{attribute 'Tc2GvlVarNames'}
VAR_GLOBAL
	{attribute 'OPC.UA.DA' := '1'}
	{attribute 'OPC.UA.DA.StructuredType' := '1'}
	arrScadaAlarms : ARRAY [1..222]  OF ST_AliasAlarms;	
	
	{attribute 'OPC.UA.DA' := '1'}
	{attribute 'OPC.UA.DA.StructuredType' := '1'}
	arrOPCUA_Alarms : ARRAY [1..10]  OF ST_Alarm_State_Alias;	
	
	
END_VAR
(*
VAR_GLOBAL PERSISTENT
stOperAlarmIniFileName: STRING:='Copy of Alarms_AR2000.xls 041121';
arrAlarmsOld: ARRAY [1..222] OF ST_AlarmStructure;
arrAlarmsOriginal,arrAlarms: ARRAY [1..222] OF ST_AlarmStructure :=[
( sName := 'a_bOperMaStInitSt', sClearName := '', sID := '1001', a := FALSE, b := FALSE, iGroup :=1, iSetDelay :=0, iResetDelay := 100, eResetMode := MANU, eBrakeProgram := B100, eAlarmProgram := 0, Enable := TRUE, iRepetitionNumber := 0 , iRepetitionPeriod := 10, Comment := 'Turbine Initialising', Param1 := (Set:=0, SetMin:=0, SetMax:=0,Comment:=''), Param2 := (Set:=0, SetMin:=0, SetMax:=0,Comment:='') ),
( sName := 'a_bOperMaStStopSt', sClearName := '', sID := '1002', a := FALSE, b := FALSE, iGroup :=1, iSetDelay :=0, iResetDelay := 0, eResetMode := MANU, eBrakeProgram := B100, eAlarmProgram := 0, Enable := TRUE, iRepetitionNumber := 0 , iRepetitionPeriod := 10, Comment := 'Turbine in the Stop state', Param1 := (Set:=0, SetMin:=0, SetMax:=0,Comment:=''), Param2 := (Set:=0, SetMin:=0, SetMax:=0,Comment:='') ),
( sName := 'a_bOperMaStIdleSt', sClearName := '', sID := '1003', a := FALSE, b := FALSE, iGroup :=1, iSetDelay :=0, iResetDelay := 0, eResetMode := MANU, eBrakeProgram := B100, eAlarmProgram := 0, Enable := TRUE, iRepetitionNumber := 0 , iRepetitionPeriod := 10, Comment := 'Turbine in the Idle state', Param1 := (Set:=0, SetMin:=0, SetMax:=0,Comment:=''), Param2 := (Set:=0, SetMin:=0, SetMax:=0,Comment:='') ),
( sName := 'a_bOperMaStStandbySt', sClearName := '', sID := '1004', a := FALSE, b := FALSE, iGroup :=1, iSetDelay :=0, iResetDelay := 0, eResetMode := MANU, eBrakeProgram := B100, eAlarmProgram := 0, Enable := TRUE, iRepetitionNumber := 0 , iRepetitionPeriod := 10, Comment := 'Turbine in the Ready state', Param1 := (Set:=0, SetMin:=0, SetMax:=0,Comment:=''), Param2 := (Set:=0, SetMin:=0, SetMax:=0,Comment:='') ),
( sName := 'a_bOperMaStPowerProductionSt', sClearName := '', sID := '1005', a := FALSE, b := FALSE, iGroup :=1, iSetDelay :=0, iResetDelay := 0, eResetMode := MANU, eBrakeProgram := B100, eAlarmProgram := 0, Enable := TRUE, iRepetitionNumber := 0 , iRepetitionPeriod := 10, Comment := 'Turbine in the Power Production state', Param1 := (Set:=0, SetMin:=0, SetMax:=0,Comment:=''), Param2 := (Set:=0, SetMin:=0, SetMax:=0,Comment:='') ),
( sName := 'a_bOperMaStNormalStopSt', sClearName := '', sID := '1006', a := FALSE, b := FALSE, iGroup :=1, iSetDelay :=0, iResetDelay := 0, eResetMode := MANU, eBrakeProgram := B100, eAlarmProgram := 0, Enable := TRUE, iRepetitionNumber := 0 , iRepetitionPeriod := 10, Comment := 'Turbine in the Normal Stop state', Param1 := (Set:=0, SetMin:=0, SetMax:=0,Comment:=''), Param2 := (Set:=0, SetMin:=0, SetMax:=0,Comment:='') ),
( sName := 'a_bOperMaStEmergencyStopSt', sClearName := '', sID := '1007', a := FALSE, b := FALSE, iGroup :=1, iSetDelay :=0, iResetDelay := 0, eResetMode := MANU, eBrakeProgram := B100, eAlarmProgram := 0, Enable := TRUE, iRepetitionNumber := 0 , iRepetitionPeriod := 10, Comment := 'Turbine in the Emergency Stop state', Param1 := (Set:=0, SetMin:=0, SetMax:=0,Comment:=''), Param2 := (Set:=0, SetMin:=0, SetMax:=0,Comment:='') ),
( sName := 'a_bOperAutostartCmdActive', sClearName := '', sID := '1008', a := FALSE, b := FALSE, iGroup :=1, iSetDelay :=0, iResetDelay := 0, eResetMode := MANU, eBrakeProgram := B99, eAlarmProgram := 0, Enable := TRUE, iRepetitionNumber := 0 , iRepetitionPeriod := 0, Comment := 'System generation inhibit removed by operator', Param1 := (Set:=0, SetMin:=0, SetMax:=0,Comment:=''), Param2 := (Set:=0, SetMin:=0, SetMax:=0,Comment:='') ),
( sName := 'a_bOperTestIdlingShutdown', sClearName := '', sID := '1009', a := FALSE, b := FALSE, iGroup :=1, iSetDelay :=0, iResetDelay := 0, eResetMode := MANU, eBrakeProgram := B17, eAlarmProgram := 0, Enable := TRUE, iRepetitionNumber := 0 , iRepetitionPeriod := 0, Comment := 'Test B17 go to Idle or Standby', Param1 := (Set:=0, SetMin:=0, SetMax:=0,Comment:=''), Param2 := (Set:=0, SetMin:=0, SetMax:=0,Comment:='') ),
( sName := 'a_bOperTestBrakingShutdown', sClearName := '', sID := '1010', a := FALSE, b := FALSE, iGroup :=1, iSetDelay :=0, iResetDelay := 0, eResetMode := MANU, eBrakeProgram := B14, eAlarmProgram := 0, Enable := TRUE, iRepetitionNumber := 0 , iRepetitionPeriod := 0, Comment := 'Test B14 apply parking brake', Param1 := (Set:=0, SetMin:=0, SetMax:=0,Comment:=''), Param2 := (Set:=0, SetMin:=0, SetMax:=0,Comment:='') ),
( sName := 'a_bOperTestSafetyVCTripShutdown', sClearName := '', sID := '1011', a := FALSE, b := FALSE, iGroup :=1, iSetDelay :=0, iResetDelay := 0, eResetMode := MANU, eBrakeProgram := B100, eAlarmProgram := 0, Enable := TRUE, iRepetitionNumber := 0 , iRepetitionPeriod := 0, Comment := 'Test B9 trip vacuum contactor', Param1 := (Set:=0, SetMin:=0, SetMax:=0,Comment:=''), Param2 := (Set:=0, SetMin:=0, SetMax:=0,Comment:='') ),
( sName := 'a_bOperTestSafetyBrakeShutdown', sClearName := '', sID := '1012', a := FALSE, b := FALSE, iGroup :=1, iSetDelay :=0, iResetDelay := 0, eResetMode := MANU, eBrakeProgram := B100, eAlarmProgram := 0, Enable := TRUE, iRepetitionNumber := 0 , iRepetitionPeriod := 0, Comment := 'Test B5 apply safety brake', Param1 := (Set:=0, SetMin:=0, SetMax:=0,Comment:=''), Param2 := (Set:=0, SetMin:=0, SetMax:=0,Comment:='') ),
( sName := 'a_bOperCmdNormalShutdownToStop', sClearName := 'Turbine manual stop using main gui button', sID := '1013', a := FALSE, b := FALSE, iGroup :=1, iSetDelay :=0, iResetDelay := 0, eResetMode := MANU, eBrakeProgram := B100, eAlarmProgram := 0, Enable := TRUE, iRepetitionNumber := 0 , iRepetitionPeriod := 0, Comment := 'Manual stop command', Param1 := (Set:=0, SetMin:=0, SetMax:=0,Comment:=''), Param2 := (Set:=0, SetMin:=0, SetMax:=0,Comment:='') ),
( sName := 'a_bOperCmdNormalShutdownToStandby', sClearName := '', sID := '1014', a := FALSE, b := FALSE, iGroup :=1, iSetDelay :=0, iResetDelay := 0, eResetMode := MANU, eBrakeProgram := B100, eAlarmProgram := 0, Enable := TRUE, iRepetitionNumber := 0 , iRepetitionPeriod := 0, Comment := '', Param1 := (Set:=0, SetMin:=0, SetMax:=0,Comment:=''), Param2 := (Set:=0, SetMin:=0, SetMax:=0,Comment:='') ),
( sName := 'a_bOperRepeatingAlarm', sClearName := '', sID := '1015', a := FALSE, b := FALSE, iGroup :=1, iSetDelay :=10, iResetDelay := 0, eResetMode := MANU, eBrakeProgram := B100, eAlarmProgram := 0, Enable := TRUE, iRepetitionNumber := 0 , iRepetitionPeriod := 10, Comment := 'Alarm which occur with this one has occured too many times', Param1 := (Set:=0, SetMin:=0, SetMax:=0,Comment:=''), Param2 := (Set:=0, SetMin:=0, SetMax:=0,Comment:='') ),
( sName := 'a_bOperResetTooLongPushed', sClearName := 'Reset Button ', sID := '1016', a := FALSE, b := FALSE, iGroup :=1, iSetDelay :=10, iResetDelay := 0, eResetMode := MANU, eBrakeProgram := B99, eAlarmProgram := 0, Enable := TRUE, iRepetitionNumber := 0 , iRepetitionPeriod := 10, Comment := 'Reset button pressed too long', Param1 := (Set:=0, SetMin:=0, SetMax:=0,Comment:=''), Param2 := (Set:=0, SetMin:=0, SetMax:=0,Comment:='') ),
( sName := 'a_bOperAlarmParameterChanged', sClearName := 'Alarm Parameter ', sID := '1017', a := FALSE, b := FALSE, iGroup :=1, iSetDelay :=0, iResetDelay := 5, eResetMode := MANU, eBrakeProgram := B99, eAlarmProgram := 0, Enable := TRUE, iRepetitionNumber := 0 , iRepetitionPeriod := 10, Comment := 'Alarm parameter has been changed', Param1 := (Set:=0, SetMin:=0, SetMax:=0,Comment:=''), Param2 := (Set:=0, SetMin:=0, SetMax:=0,Comment:='') ),
( sName := 'a_bOperIniParameterChanged', sClearName := 'Ini Parameter ', sID := '1018', a := FALSE, b := FALSE, iGroup :=1, iSetDelay :=0, iResetDelay := 5, eResetMode := MANU, eBrakeProgram := B99, eAlarmProgram := 0, Enable := TRUE, iRepetitionNumber := 0 , iRepetitionPeriod := 10, Comment := 'Ini parameter has been changed', Param1 := (Set:=0, SetMin:=0, SetMax:=0,Comment:=''), Param2 := (Set:=0, SetMin:=0, SetMax:=0,Comment:='') ),
( sName := 'a_bOperSystemReboot', sClearName := 'System ', sID := '1019', a := FALSE, b := FALSE, iGroup :=1, iSetDelay :=10, iResetDelay := 150, eResetMode := MANU, eBrakeProgram := B100, eAlarmProgram := 0, Enable := TRUE, iRepetitionNumber := 0 , iRepetitionPeriod := 10, Comment := 'System is rebooted', Param1 := (Set:=0, SetMin:=0, SetMax:=0,Comment:=''), Param2 := (Set:=0, SetMin:=0, SetMax:=0,Comment:='') ),
( sName := 'a_bOperSystemRestart ', sClearName := 'System ', sID := '1020', a := FALSE, b := FALSE, iGroup :=1, iSetDelay :=10, iResetDelay := 150, eResetMode := MANU, eBrakeProgram := B100, eAlarmProgram := 0, Enable := TRUE, iRepetitionNumber := 0 , iRepetitionPeriod := 10, Comment := 'System is restarted', Param1 := (Set:=0, SetMin:=0, SetMax:=0,Comment:=''), Param2 := (Set:=0, SetMin:=0, SetMax:=0,Comment:='') ),
( sName := 'a_bOperScopeViewNotActive', sClearName := 'ScopeView running', sID := '1021', a := FALSE, b := FALSE, iGroup :=1, iSetDelay :=100, iResetDelay := 0, eResetMode := MANU, eBrakeProgram := B17, eAlarmProgram := 0, Enable := TRUE, iRepetitionNumber := 0 , iRepetitionPeriod := 10, Comment := 'Fastlog system not active', Param1 := (Set:=0, SetMin:=0, SetMax:=0,Comment:=''), Param2 := (Set:=0, SetMin:=0, SetMax:=0,Comment:='') ),
( sName := 'a_bOperXMLDataUncertainty', sClearName := 'Turbine data XML file Ok', sID := '1022', a := FALSE, b := FALSE, iGroup :=1, iSetDelay :=0, iResetDelay := 0, eResetMode := MANU, eBrakeProgram := B17, eAlarmProgram := 0, Enable := TRUE, iRepetitionNumber := 0 , iRepetitionPeriod := 10, Comment := 'Turbine data XML file uncertainty', Param1 := (Set:=0, SetMin:=0, SetMax:=0,Comment:=''), Param2 := (Set:=0, SetMin:=0, SetMax:=0,Comment:='') ),
( sName := 'a_bOperSoftwareUpdate', sClearName := 'System software ', sID := '1023', a := FALSE, b := FALSE, iGroup :=1, iSetDelay :=0, iResetDelay := 0, eResetMode := MANU, eBrakeProgram := B17, eAlarmProgram := 0, Enable := FALSE, iRepetitionNumber := 0 , iRepetitionPeriod := 10, Comment := 'System software is updated', Param1 := (Set:=0, SetMin:=0, SetMax:=0,Comment:=''), Param2 := (Set:=0, SetMin:=0, SetMax:=0,Comment:='') ),
( sName := 'a_bOperFastlogComsErr', sClearName := 'a_bOperLossOfCommsToArrayController', sID := '1024', a := FALSE, b := FALSE, iGroup :=1, iSetDelay :=0, iResetDelay := 0, eResetMode := MANU, eBrakeProgram := B99, eAlarmProgram := 0, Enable := TRUE, iRepetitionNumber := 0 , iRepetitionPeriod := 10, Comment := 'Loss of Comms with ARL Array PLC', Param1 := (Set:=0, SetMin:=0, SetMax:=0,Comment:=''), Param2 := (Set:=0, SetMin:=0, SetMax:=0,Comment:='') ),
( sName := 'a_bOperInOffMode', sClearName := 'Turbine in OFF Mode', sID := '1025', a := FALSE, b := FALSE, iGroup :=1, iSetDelay :=0, iResetDelay := 0, eResetMode := MANU, eBrakeProgram := B100, eAlarmProgram := 0, Enable := TRUE, iRepetitionNumber := 0 , iRepetitionPeriod := 10, Comment := 'Turbine entering OFF Mode', Param1 := (Set:=0, SetMin:=0, SetMax:=0,Comment:=''), Param2 := (Set:=0, SetMin:=0, SetMax:=0,Comment:='') ),
( sName := 'a_bOperInServiceMode', sClearName := 'Turbine in Service Mode', sID := '1026', a := FALSE, b := FALSE, iGroup :=1, iSetDelay :=0, iResetDelay := 0, eResetMode := MANU, eBrakeProgram := B100, eAlarmProgram := 0, Enable := TRUE, iRepetitionNumber := 0 , iRepetitionPeriod := 10, Comment := 'Turbine entering Service Mode', Param1 := (Set:=0, SetMin:=0, SetMax:=0,Comment:=''), Param2 := (Set:=0, SetMin:=0, SetMax:=0,Comment:='') ),
( sName := 'a_bOperInAutomaticMode', sClearName := 'Turbine in Automatic Mode', sID := '1027', a := FALSE, b := FALSE, iGroup :=1, iSetDelay :=0, iResetDelay := 0, eResetMode := MANU, eBrakeProgram := B100, eAlarmProgram := 0, Enable := TRUE, iRepetitionNumber := 0 , iRepetitionPeriod := 10, Comment := 'Turbine entering Automatic Mode', Param1 := (Set:=0, SetMin:=0, SetMax:=0,Comment:=''), Param2 := (Set:=0, SetMin:=0, SetMax:=0,Comment:='') ),
( sName := 'a_bOperInManualMode', sClearName := 'Turbine in Manual Mode', sID := '1028', a := FALSE, b := FALSE, iGroup :=1, iSetDelay :=0, iResetDelay := 0, eResetMode := MANU, eBrakeProgram := B100, eAlarmProgram := 0, Enable := TRUE, iRepetitionNumber := 0 , iRepetitionPeriod := 10, Comment := 'Turbine entering Manual Mode', Param1 := (Set:=0, SetMin:=0, SetMax:=0,Comment:=''), Param2 := (Set:=0, SetMin:=0, SetMax:=0,Comment:='') ),
( sName := 'a_bOperInFATMode', sClearName := 'Turbine in Factory Acceptance Test Nautilus Mode', sID := '1029', a := FALSE, b := FALSE, iGroup :=1, iSetDelay :=0, iResetDelay := 0, eResetMode := MANU, eBrakeProgram := B100, eAlarmProgram := 0, Enable := TRUE, iRepetitionNumber := 0 , iRepetitionPeriod := 10, Comment := 'Turbine entering Factory Acceptance Test Nautilus Mode', Param1 := (Set:=0, SetMin:=0, SetMax:=0,Comment:=''), Param2 := (Set:=0, SetMin:=0, SetMax:=0,Comment:='') ),
( sName := 'a_bHydairFaultActive', sClearName := 'Cleared', sID := '1030', a := FALSE, b := FALSE, iGroup :=1, iSetDelay :=0, iResetDelay := 0, eResetMode := MANU, eBrakeProgram := B99, eAlarmProgram := 0, Enable := TRUE, iRepetitionNumber := 0 , iRepetitionPeriod := 0, Comment := '', Param1 := (Set:=0, SetMin:=0, SetMax:=0,Comment:=''), Param2 := (Set:=0, SetMin:=0, SetMax:=0,Comment:='') ),
( sName := 'a_bHydairOfflineFilterClogged', sClearName := 'Cleared', sID := '1031', a := FALSE, b := FALSE, iGroup :=1, iSetDelay :=0, iResetDelay := 0, eResetMode := MANU, eBrakeProgram := B99, eAlarmProgram := 0, Enable := TRUE, iRepetitionNumber := 0 , iRepetitionPeriod := 0, Comment := '', Param1 := (Set:=0, SetMin:=0, SetMax:=0,Comment:=''), Param2 := (Set:=0, SetMin:=0, SetMax:=0,Comment:='') ),
( sName := 'a_bMainReturnPressureFilterClogged', sClearName := 'Cleared', sID := '1032', a := FALSE, b := FALSE, iGroup :=1, iSetDelay :=0, iResetDelay := 0, eResetMode := MANU, eBrakeProgram := B99, eAlarmProgram := 0, Enable := TRUE, iRepetitionNumber := 0 , iRepetitionPeriod := 0, Comment := '', Param1 := (Set:=0, SetMin:=0, SetMax:=0,Comment:=''), Param2 := (Set:=0, SetMin:=0, SetMax:=0,Comment:='') ),
( sName := 'a_bMainSupplyPressureFilterClogged', sClearName := 'Cleared', sID := '1033', a := FALSE, b := FALSE, iGroup :=1, iSetDelay :=0, iResetDelay := 0, eResetMode := MANU, eBrakeProgram := B99, eAlarmProgram := 0, Enable := TRUE, iRepetitionNumber := 0 , iRepetitionPeriod := 0, Comment := '', Param1 := (Set:=0, SetMin:=0, SetMax:=0,Comment:=''), Param2 := (Set:=0, SetMin:=0, SetMax:=0,Comment:='') ),
( sName := 'a_bHydairPassiveCtrlState', sClearName := 'Cleared', sID := '1034', a := FALSE, b := FALSE, iGroup :=1, iSetDelay :=0, iResetDelay := 0, eResetMode := MANU, eBrakeProgram := B99, eAlarmProgram := 0, Enable := TRUE, iRepetitionNumber := 0 , iRepetitionPeriod := 0, Comment := '', Param1 := (Set:=0, SetMin:=0, SetMax:=0,Comment:=''), Param2 := (Set:=0, SetMin:=0, SetMax:=0,Comment:='') ),
( sName := 'a_bHydairStartUp', sClearName := 'Cleared', sID := '1035', a := FALSE, b := FALSE, iGroup :=1, iSetDelay :=0, iResetDelay := 0, eResetMode := MANU, eBrakeProgram := B99, eAlarmProgram := 0, Enable := TRUE, iRepetitionNumber := 0 , iRepetitionPeriod := 0, Comment := '', Param1 := (Set:=0, SetMin:=0, SetMax:=0,Comment:=''), Param2 := (Set:=0, SetMin:=0, SetMax:=0,Comment:='') ),
( sName := 'a_bHydairReadyToOperate', sClearName := 'Cleared', sID := '1036', a := FALSE, b := FALSE, iGroup :=1, iSetDelay :=0, iResetDelay := 0, eResetMode := MANU, eBrakeProgram := B99, eAlarmProgram := 0, Enable := TRUE, iRepetitionNumber := 0 , iRepetitionPeriod := 0, Comment := '', Param1 := (Set:=0, SetMin:=0, SetMax:=0,Comment:=''), Param2 := (Set:=0, SetMin:=0, SetMax:=0,Comment:='') ),
( sName := 'a_bHydairActiveCtrlState', sClearName := 'Cleared', sID := '1037', a := FALSE, b := FALSE, iGroup :=1, iSetDelay :=0, iResetDelay := 0, eResetMode := MANU, eBrakeProgram := B99, eAlarmProgram := 0, Enable := TRUE, iRepetitionNumber := 0 , iRepetitionPeriod := 0, Comment := '', Param1 := (Set:=0, SetMin:=0, SetMax:=0,Comment:=''), Param2 := (Set:=0, SetMin:=0, SetMax:=0,Comment:='') ),
( sName := 'a_bHydairStopped', sClearName := 'Cleared', sID := '1038', a := FALSE, b := FALSE, iGroup :=1, iSetDelay :=0, iResetDelay := 0, eResetMode := MANU, eBrakeProgram := B99, eAlarmProgram := 0, Enable := TRUE, iRepetitionNumber := 0 , iRepetitionPeriod := 0, Comment := '', Param1 := (Set:=0, SetMin:=0, SetMax:=0,Comment:=''), Param2 := (Set:=0, SetMin:=0, SetMax:=0,Comment:='') ),
( sName := 'a_bHydairEstopActive', sClearName := 'Cleared', sID := '1039', a := FALSE, b := FALSE, iGroup :=1, iSetDelay :=0, iResetDelay := 0, eResetMode := MANU, eBrakeProgram := B99, eAlarmProgram := 0, Enable := TRUE, iRepetitionNumber := 0 , iRepetitionPeriod := 0, Comment := '', Param1 := (Set:=0, SetMin:=0, SetMax:=0,Comment:=''), Param2 := (Set:=0, SetMin:=0, SetMax:=0,Comment:='') ),
( sName := 'a_bHydairOilTempTooHigh', sClearName := 'Cleared', sID := '1040', a := FALSE, b := FALSE, iGroup :=1, iSetDelay :=0, iResetDelay := 0, eResetMode := MANU, eBrakeProgram := B99, eAlarmProgram := 0, Enable := TRUE, iRepetitionNumber := 0 , iRepetitionPeriod := 0, Comment := '', Param1 := (Set:=0, SetMin:=0, SetMax:=0,Comment:=''), Param2 := (Set:=0, SetMin:=0, SetMax:=0,Comment:='') ),
( sName := 'a_bHydairReadyToStartup', sClearName := 'Cleared', sID := '1041', a := FALSE, b := FALSE, iGroup :=1, iSetDelay :=0, iResetDelay := 0, eResetMode := MANU, eBrakeProgram := B99, eAlarmProgram := 0, Enable := TRUE, iRepetitionNumber := 0 , iRepetitionPeriod := 0, Comment := '', Param1 := (Set:=0, SetMin:=0, SetMax:=0,Comment:=''), Param2 := (Set:=0, SetMin:=0, SetMax:=0,Comment:='') ),
( sName := 'a_bOperRequestStopLATSystem', sClearName := 'Cleared', sID := '1042', a := FALSE, b := FALSE, iGroup :=1, iSetDelay :=0, iResetDelay := 0, eResetMode := MANU, eBrakeProgram := B99, eAlarmProgram := 0, Enable := TRUE, iRepetitionNumber := 0 , iRepetitionPeriod := 0, Comment := '', Param1 := (Set:=0, SetMin:=0, SetMax:=0,Comment:=''), Param2 := (Set:=0, SetMin:=0, SetMax:=0,Comment:='') ),
( sName := 'a_bOperRequestStartupHydair', sClearName := 'Cleared', sID := '1043', a := FALSE, b := FALSE, iGroup :=1, iSetDelay :=0, iResetDelay := 0, eResetMode := MANU, eBrakeProgram := B99, eAlarmProgram := 0, Enable := TRUE, iRepetitionNumber := 0 , iRepetitionPeriod := 0, Comment := '', Param1 := (Set:=0, SetMin:=0, SetMax:=0,Comment:=''), Param2 := (Set:=0, SetMin:=0, SetMax:=0,Comment:='') ),
( sName := 'a_bOperRequestPassivePitchCtrl', sClearName := 'Cleared', sID := '1044', a := FALSE, b := FALSE, iGroup :=1, iSetDelay :=0, iResetDelay := 0, eResetMode := MANU, eBrakeProgram := B99, eAlarmProgram := 0, Enable := TRUE, iRepetitionNumber := 0 , iRepetitionPeriod := 0, Comment := '', Param1 := (Set:=0, SetMin:=0, SetMax:=0,Comment:=''), Param2 := (Set:=0, SetMin:=0, SetMax:=0,Comment:='') ),
( sName := 'a_bOperRequestActiveLoadCtrlMode', sClearName := 'Cleared', sID := '1045', a := FALSE, b := FALSE, iGroup :=1, iSetDelay :=0, iResetDelay := 0, eResetMode := MANU, eBrakeProgram := B99, eAlarmProgram := 0, Enable := TRUE, iRepetitionNumber := 0 , iRepetitionPeriod := 0, Comment := '', Param1 := (Set:=0, SetMin:=0, SetMax:=0,Comment:=''), Param2 := (Set:=0, SetMin:=0, SetMax:=0,Comment:='') ),
( sName := 'a_bOperRequestLoadProfileStream', sClearName := 'Cleared', sID := '1046', a := FALSE, b := FALSE, iGroup :=1, iSetDelay :=0, iResetDelay := 0, eResetMode := MANU, eBrakeProgram := B99, eAlarmProgram := 0, Enable := TRUE, iRepetitionNumber := 0 , iRepetitionPeriod := 0, Comment := '', Param1 := (Set:=0, SetMin:=0, SetMax:=0,Comment:=''), Param2 := (Set:=0, SetMin:=0, SetMax:=0,Comment:='') ),
( sName := 'a_bOperLoadProfileStreamingStarted', sClearName := 'Cleared', sID := '1047', a := FALSE, b := FALSE, iGroup :=1, iSetDelay :=0, iResetDelay := 0, eResetMode := MANU, eBrakeProgram := B99, eAlarmProgram := 0, Enable := TRUE, iRepetitionNumber := 0 , iRepetitionPeriod := 0, Comment := '', Param1 := (Set:=0, SetMin:=0, SetMax:=0,Comment:=''), Param2 := (Set:=0, SetMin:=0, SetMax:=0,Comment:='') ),
( sName := 'a_bOperLoadProfilePaused', sClearName := 'Cleared', sID := '1048', a := FALSE, b := FALSE, iGroup :=1, iSetDelay :=0, iResetDelay := 0, eResetMode := MANU, eBrakeProgram := B99, eAlarmProgram := 0, Enable := TRUE, iRepetitionNumber := 0 , iRepetitionPeriod := 0, Comment := '', Param1 := (Set:=0, SetMin:=0, SetMax:=0,Comment:=''), Param2 := (Set:=0, SetMin:=0, SetMax:=0,Comment:='') ),
( sName := 'a_bOperLoadProfileFrequencyError', sClearName := 'Cleared', sID := '1049', a := FALSE, b := FALSE, iGroup :=1, iSetDelay :=0, iResetDelay := 0, eResetMode := MANU, eBrakeProgram := B99, eAlarmProgram := 0, Enable := TRUE, iRepetitionNumber := 0 , iRepetitionPeriod := 0, Comment := '', Param1 := (Set:=0, SetMin:=0, SetMax:=0,Comment:=''), Param2 := (Set:=0, SetMin:=0, SetMax:=0,Comment:='') ),
( sName := 'a_bOperPitch100HrRuntime', sClearName := 'Cleared', sID := '1050', a := FALSE, b := FALSE, iGroup :=1, iSetDelay :=0, iResetDelay := 0, eResetMode := MANU, eBrakeProgram := B99, eAlarmProgram := 0, Enable := TRUE, iRepetitionNumber := 0 , iRepetitionPeriod := 0, Comment := '', Param1 := (Set:=0, SetMin:=0, SetMax:=0,Comment:=''), Param2 := (Set:=0, SetMin:=0, SetMax:=0,Comment:='') ),
( sName := 'a_bOperB20PitchNormalShutdownCmd', sClearName := 'Cleared', sID := '1051', a := FALSE, b := FALSE, iGroup :=1, iSetDelay :=0, iResetDelay := 0, eResetMode := MANU, eBrakeProgram := B20, eAlarmProgram := 0, Enable := TRUE, iRepetitionNumber := 0 , iRepetitionPeriod := 0, Comment := '', Param1 := (Set:=0, SetMin:=0, SetMax:=0,Comment:=''), Param2 := (Set:=0, SetMin:=0, SetMax:=0,Comment:='') ),
( sName := 'a_bHydraulicsLoadMzRam1HiWarning', sClearName := 'Hydraulic Load Hi Warning', sID := '1045', a := FALSE, b := FALSE, iGroup :=1, iSetDelay :=0, iResetDelay := 0, eResetMode := MANU, eBrakeProgram := B20, eAlarmProgram := 0, Enable := TRUE, iRepetitionNumber := 0 , iRepetitionPeriod := 0, Comment := 'Hydraulic Load Hi Warning', Param1 := (Set:=450000, SetMin:=1, SetMax:=600000,Comment:='Nm'), Param2 := (Set:=1000, SetMin:=1, SetMax:=600000,Comment:='Nm') ),
( sName := 'a_bHydraulicsLoadMzRam1HiHiAlarm', sClearName := 'Hydraulic Load Hi Alarm', sID := '1046', a := FALSE, b := FALSE, iGroup :=1, iSetDelay :=0, iResetDelay := 0, eResetMode := MANU, eBrakeProgram := B1, eAlarmProgram := 0, Enable := TRUE, iRepetitionNumber := 0 , iRepetitionPeriod := 0, Comment := 'Hydraulic Load Hi Alarm', Param1 := (Set:=500000, SetMin:=1, SetMax:=600000,Comment:='Nm'), Param2 := (Set:=1000, SetMin:=1, SetMax:=600000,Comment:='Nm') ),
( sName := 'a_bHydraulicsLoadMyRam2HiWarning', sClearName := 'Hydraulic Load Hi Warning', sID := '1047', a := FALSE, b := FALSE, iGroup :=1, iSetDelay :=0, iResetDelay := 0, eResetMode := MANU, eBrakeProgram := B20, eAlarmProgram := 0, Enable := TRUE, iRepetitionNumber := 0 , iRepetitionPeriod := 0, Comment := 'Hydraulic Load Hi Warning', Param1 := (Set:=450000, SetMin:=1, SetMax:=600000,Comment:='Nm'), Param2 := (Set:=1000, SetMin:=1, SetMax:=600000,Comment:='Nm') ),
( sName := 'a_bHydraulicsLoadMyRam2HiHiAlarm', sClearName := 'Hydraulic Load Hi Alarm', sID := '1048', a := FALSE, b := FALSE, iGroup :=1, iSetDelay :=0, iResetDelay := 0, eResetMode := MANU, eBrakeProgram := B1, eAlarmProgram := 0, Enable := TRUE, iRepetitionNumber := 0 , iRepetitionPeriod := 0, Comment := 'Hydraulic Load Hi Alarm', Param1 := (Set:=500000, SetMin:=1, SetMax:=600000,Comment:='Nm'), Param2 := (Set:=1000, SetMin:=1, SetMax:=600000,Comment:='Nm') ),
( sName := 'a_bHydraulicsLoadTrackingMzRAM1Warning', sClearName := 'Hydraulic Load Control Tracking Warning', sID := '1049', a := FALSE, b := FALSE, iGroup :=1, iSetDelay :=10, iResetDelay := 10, eResetMode := MANU, eBrakeProgram := B99, eAlarmProgram := 0, Enable := TRUE, iRepetitionNumber := 0 , iRepetitionPeriod := 0, Comment := 'Hydraulic Load Control Tracking Warning', Param1 := (Set:=5, SetMin:=0, SetMax:=100,Comment:=''), Param2 := (Set:=2, SetMin:=0, SetMax:=100,Comment:='') ),
( sName := 'a_bHydraulicsLoadTrackingMzRAM1Alarm', sClearName := 'Hydraulic Load Control Tracking Alarm', sID := '1050', a := FALSE, b := FALSE, iGroup :=1, iSetDelay :=10, iResetDelay := 10, eResetMode := MANU, eBrakeProgram := B20, eAlarmProgram := 0, Enable := TRUE, iRepetitionNumber := 0 , iRepetitionPeriod := 0, Comment := 'Hydraulic Load Control Tracking Alarm', Param1 := (Set:=10, SetMin:=0, SetMax:=100,Comment:=''), Param2 := (Set:=5, SetMin:=0, SetMax:=100,Comment:='') ),
( sName := 'a_bHydraulicsLoadTrackingMyRAM2Warning', sClearName := 'Hydraulic Load Control Tracking Warning', sID := '1051', a := FALSE, b := FALSE, iGroup :=1, iSetDelay :=10, iResetDelay := 10, eResetMode := MANU, eBrakeProgram := B99, eAlarmProgram := 0, Enable := TRUE, iRepetitionNumber := 0 , iRepetitionPeriod := 0, Comment := 'Hydraulic Load Control Tracking Warning', Param1 := (Set:=5, SetMin:=0, SetMax:=100,Comment:=''), Param2 := (Set:=2, SetMin:=0, SetMax:=100,Comment:='') ),
( sName := 'a_bHydraulicsLoadTrackingMyRAM2Alarm', sClearName := 'Hydraulic Load Control Tracking Alarm', sID := '1052', a := FALSE, b := FALSE, iGroup :=1, iSetDelay :=10, iResetDelay := 10, eResetMode := MANU, eBrakeProgram := B20, eAlarmProgram := 0, Enable := TRUE, iRepetitionNumber := 0 , iRepetitionPeriod := 0, Comment := 'Hydraulic Load Control Tracking Alarm', Param1 := (Set:=10, SetMin:=0, SetMax:=100,Comment:=''), Param2 := (Set:=5, SetMin:=0, SetMax:=100,Comment:='') ),
( sName := 'a_bHydraulicsLVDTSensor1Failure', sClearName := 'Hydraulics LVDT Sensor1 Failure', sID := '1053', a := FALSE, b := FALSE, iGroup :=1, iSetDelay :=0, iResetDelay := 10, eResetMode := MANU, eBrakeProgram := B99, eAlarmProgram := 0, Enable := TRUE, iRepetitionNumber := 0 , iRepetitionPeriod := , Comment := 'Hydraulics LVDT Sensor1 Failure', Param1 := (Set:=0, SetMin:=0, SetMax:=0,Comment:=''), Param2 := (Set:=0, SetMin:=0, SetMax:=0,Comment:='') ),
( sName := 'a_bHydraulicsLVDTSensor2Failure', sClearName := 'Hydraulics LVDT Sensor2 Failure', sID := '1054', a := FALSE, b := FALSE, iGroup :=1, iSetDelay :=0, iResetDelay := 10, eResetMode := MANU, eBrakeProgram := B99, eAlarmProgram := 0, Enable := TRUE, iRepetitionNumber := 0 , iRepetitionPeriod := , Comment := 'Hydraulics LVDT Sensor2 Failure', Param1 := (Set:=0, SetMin:=0, SetMax:=0,Comment:=''), Param2 := (Set:=0, SetMin:=0, SetMax:=0,Comment:='') ),
( sName := 'a_bHydraulicsLVDTSensor3Failure', sClearName := 'Hydraulics LVDT Sensor3 Failure', sID := '1055', a := FALSE, b := FALSE, iGroup :=1, iSetDelay :=0, iResetDelay := 10, eResetMode := MANU, eBrakeProgram := B99, eAlarmProgram := 0, Enable := TRUE, iRepetitionNumber := 0 , iRepetitionPeriod := , Comment := 'Hydraulics LVDT Sensor3 Failure', Param1 := (Set:=0, SetMin:=0, SetMax:=0,Comment:=''), Param2 := (Set:=0, SetMin:=0, SetMax:=0,Comment:='') ),
( sName := 'a_bHydraulicsLVDTSensor4Failure', sClearName := 'Hydraulics LVDT Sensor4 Failure', sID := '1056', a := FALSE, b := FALSE, iGroup :=1, iSetDelay :=0, iResetDelay := 10, eResetMode := MANU, eBrakeProgram := B99, eAlarmProgram := 0, Enable := TRUE, iRepetitionNumber := 0 , iRepetitionPeriod := , Comment := 'Hydraulics LVDT Sensor4 Failure', Param1 := (Set:=0, SetMin:=0, SetMax:=0,Comment:=''), Param2 := (Set:=0, SetMin:=0, SetMax:=0,Comment:='') ),
( sName := 'a_bHydraulicsLVDTSensor5Failure', sClearName := 'Hydraulics LVDT Sensor5 Failure', sID := '1057', a := FALSE, b := FALSE, iGroup :=1, iSetDelay :=0, iResetDelay := 10, eResetMode := MANU, eBrakeProgram := B99, eAlarmProgram := 0, Enable := TRUE, iRepetitionNumber := 0 , iRepetitionPeriod := , Comment := 'Hydraulics LVDT Sensor5 Failure', Param1 := (Set:=0, SetMin:=0, SetMax:=0,Comment:=''), Param2 := (Set:=0, SetMin:=0, SetMax:=0,Comment:='') ),
( sName := 'a_bHydraulicsLVDTSensor6Failure', sClearName := 'Hydraulics LVDT Sensor6 Failure', sID := '1058', a := FALSE, b := FALSE, iGroup :=1, iSetDelay :=0, iResetDelay := 10, eResetMode := MANU, eBrakeProgram := B99, eAlarmProgram := 0, Enable := TRUE, iRepetitionNumber := 0 , iRepetitionPeriod := , Comment := 'Hydraulics LVDT Sensor6 Failure', Param1 := (Set:=0, SetMin:=0, SetMax:=0,Comment:=''), Param2 := (Set:=0, SetMin:=0, SetMax:=0,Comment:='') ),
( sName := 'a_bHydraulicsLVDTSensor7Failure', sClearName := 'Hydraulics LVDT Sensor7 Failure', sID := '1059', a := FALSE, b := FALSE, iGroup :=1, iSetDelay :=0, iResetDelay := 10, eResetMode := MANU, eBrakeProgram := B99, eAlarmProgram := 0, Enable := TRUE, iRepetitionNumber := 0 , iRepetitionPeriod := , Comment := 'Hydraulics LVDT Sensor7 Failure', Param1 := (Set:=0, SetMin:=0, SetMax:=0,Comment:=''), Param2 := (Set:=0, SetMin:=0, SetMax:=0,Comment:='') ),
( sName := 'a_bHydraulicsLVDTSensor8Failure', sClearName := 'Hydraulics LVDT Sensor8 Failure', sID := '1060', a := FALSE, b := FALSE, iGroup :=1, iSetDelay :=0, iResetDelay := 10, eResetMode := MANU, eBrakeProgram := B99, eAlarmProgram := 0, Enable := TRUE, iRepetitionNumber := 0 , iRepetitionPeriod := , Comment := 'Hydraulics LVDT Sensor8 Failure', Param1 := (Set:=0, SetMin:=0, SetMax:=0,Comment:=''), Param2 := (Set:=0, SetMin:=0, SetMax:=0,Comment:='') ),
( sName := 'a_bHydraulicsMzStrainGaugeFailure', sClearName := 'Hydraulics Mz Strain Gauge Failure', sID := '1061', a := FALSE, b := FALSE, iGroup :=1, iSetDelay :=0, iResetDelay := 10, eResetMode := MANU, eBrakeProgram := B20, eAlarmProgram := 0, Enable := TRUE, iRepetitionNumber := 0 , iRepetitionPeriod := , Comment := 'a_bHydraulicsMzStrainGaugeFailure', Param1 := (Set:=0, SetMin:=0, SetMax:=0,Comment:=''), Param2 := (Set:=0, SetMin:=0, SetMax:=0,Comment:='') ),
( sName := 'a_bHydraulicsMzStrainGaugeFailure', sClearName := 'Hydraulics Mz Strain Gauge Failure', sID := '1062', a := FALSE, b := FALSE, iGroup :=1, iSetDelay :=0, iResetDelay := 10, eResetMode := MANU, eBrakeProgram := B20, eAlarmProgram := 0, Enable := TRUE, iRepetitionNumber := 0 , iRepetitionPeriod := , Comment := 'a_bHydraulicsMzStrainGaugeFailure', Param1 := (Set:=0, SetMin:=0, SetMax:=0,Comment:=''), Param2 := (Set:=0, SetMin:=0, SetMax:=0,Comment:='') ),
( sName := 'a_bSafetyCommsLossToSSB', sClearName := '', sID := '2001', a := FALSE, b := FALSE, iGroup :=2, iSetDelay :=0, iResetDelay := 0, eResetMode := MANU, eBrakeProgram := B4, eAlarmProgram := 0, Enable := TRUE, iRepetitionNumber := 0 , iRepetitionPeriod := 0, Comment := '', Param1 := (Set:=0, SetMin:=0, SetMax:=0,Comment:=''), Param2 := (Set:=0, SetMin:=0, SetMax:=0,Comment:='') ),
( sName := 'a_bSafetyEPO_Main_Panel', sClearName := '', sID := '2002', a := FALSE, b := FALSE, iGroup :=2, iSetDelay :=0, iResetDelay := 0, eResetMode := MANU, eBrakeProgram := B1, eAlarmProgram := 0, Enable := TRUE, iRepetitionNumber := 0 , iRepetitionPeriod := 0, Comment := '', Param1 := (Set:=0, SetMin:=0, SetMax:=0,Comment:=''), Param2 := (Set:=0, SetMin:=0, SetMax:=0,Comment:='') ),
( sName := 'a_bSafetyEPO_REMOTE', sClearName := '', sID := '2003', a := FALSE, b := FALSE, iGroup :=2, iSetDelay :=0, iResetDelay := 0, eResetMode := MANU, eBrakeProgram := B1, eAlarmProgram := 0, Enable := TRUE, iRepetitionNumber := 0 , iRepetitionPeriod := 0, Comment := '', Param1 := (Set:=0, SetMin:=0, SetMax:=0,Comment:=''), Param2 := (Set:=0, SetMin:=0, SetMax:=0,Comment:='') ),
( sName := 'a_bSafetyEPO_SCADA', sClearName := '', sID := '2004', a := FALSE, b := FALSE, iGroup :=2, iSetDelay :=0, iResetDelay := 0, eResetMode := MANU, eBrakeProgram := B1, eAlarmProgram := 0, Enable := TRUE, iRepetitionNumber := 0 , iRepetitionPeriod := 0, Comment := '', Param1 := (Set:=0, SetMin:=0, SetMax:=0,Comment:=''), Param2 := (Set:=0, SetMin:=0, SetMax:=0,Comment:='') ),
( sName := 'a_bSafetyEPO_TCP', sClearName := '', sID := '2005', a := FALSE, b := FALSE, iGroup :=2, iSetDelay :=0, iResetDelay := 0, eResetMode := MANU, eBrakeProgram := B1, eAlarmProgram := 0, Enable := TRUE, iRepetitionNumber := 0 , iRepetitionPeriod := 0, Comment := '', Param1 := (Set:=0, SetMin:=0, SetMax:=0,Comment:=''), Param2 := (Set:=0, SetMin:=0, SetMax:=0,Comment:='') ),
( sName := 'a_bSafetyOperatorRequestB1', sClearName := '', sID := '2006', a := FALSE, b := FALSE, iGroup :=2, iSetDelay :=0, iResetDelay := 0, eResetMode := MANU, eBrakeProgram := B1, eAlarmProgram := 0, Enable := TRUE, iRepetitionNumber := 0 , iRepetitionPeriod := 0, Comment := '', Param1 := (Set:=0, SetMin:=0, SetMax:=0,Comment:=''), Param2 := (Set:=0, SetMin:=0, SetMax:=0,Comment:='') ),
( sName := 'a_bSafetyOperatorRequestB4', sClearName := '', sID := '2007', a := FALSE, b := FALSE, iGroup :=2, iSetDelay :=0, iResetDelay := 0, eResetMode := MANU, eBrakeProgram := B4, eAlarmProgram := 0, Enable := TRUE, iRepetitionNumber := 0 , iRepetitionPeriod := 0, Comment := '', Param1 := (Set:=0, SetMin:=0, SetMax:=0,Comment:=''), Param2 := (Set:=0, SetMin:=0, SetMax:=0,Comment:='') ),
( sName := 'a_bSafetyOperatorRequestB9', sClearName := '', sID := '2008', a := FALSE, b := FALSE, iGroup :=2, iSetDelay :=0, iResetDelay := 0, eResetMode := MANU, eBrakeProgram := B9, eAlarmProgram := 0, Enable := TRUE, iRepetitionNumber := 0 , iRepetitionPeriod := 0, Comment := '', Param1 := (Set:=0, SetMin:=0, SetMax:=0,Comment:=''), Param2 := (Set:=0, SetMin:=0, SetMax:=0,Comment:='') ),
( sName := 'a_bSafetyEncoderPositionNOTValid', sClearName := '', sID := '2009', a := FALSE, b := FALSE, iGroup :=2, iSetDelay :=0, iResetDelay := 0, eResetMode := MANU, eBrakeProgram := B1, eAlarmProgram := 0, Enable := TRUE, iRepetitionNumber := 0 , iRepetitionPeriod := 0, Comment := '', Param1 := (Set:=0, SetMin:=0, SetMax:=0,Comment:=''), Param2 := (Set:=0, SetMin:=0, SetMax:=0,Comment:='') ),
( sName := 'a_bSafetyEncoderGroupError', sClearName := '', sID := '2010', a := FALSE, b := FALSE, iGroup :=2, iSetDelay :=0, iResetDelay := 0, eResetMode := MANU, eBrakeProgram := B1, eAlarmProgram := 0, Enable := TRUE, iRepetitionNumber := 0 , iRepetitionPeriod := 0, Comment := '', Param1 := (Set:=0, SetMin:=0, SetMax:=0,Comment:=''), Param2 := (Set:=0, SetMin:=0, SetMax:=0,Comment:='') ),
( sName := 'a_bSafetyIOGroupError', sClearName := '', sID := '2011', a := FALSE, b := FALSE, iGroup :=2, iSetDelay :=0, iResetDelay := 0, eResetMode := MANU, eBrakeProgram := B1, eAlarmProgram := 0, Enable := TRUE, iRepetitionNumber := 0 , iRepetitionPeriod := 0, Comment := '', Param1 := (Set:=0, SetMin:=0, SetMax:=0,Comment:=''), Param2 := (Set:=0, SetMin:=0, SetMax:=0,Comment:='') ),
( sName := 'a_bSafetyAngInGroupError', sClearName := '', sID := '2012', a := FALSE, b := FALSE, iGroup :=2, iSetDelay :=0, iResetDelay := 0, eResetMode := MANU, eBrakeProgram := B1, eAlarmProgram := 0, Enable := TRUE, iRepetitionNumber := 0 , iRepetitionPeriod := 0, Comment := '', Param1 := (Set:=0, SetMin:=0, SetMax:=0,Comment:=''), Param2 := (Set:=0, SetMin:=0, SetMax:=0,Comment:='') ),
( sName := 'a_bSafetyPresetGroupError', sClearName := '', sID := '2013', a := FALSE, b := FALSE, iGroup :=2, iSetDelay :=0, iResetDelay := 0, eResetMode := MANU, eBrakeProgram := B1, eAlarmProgram := 0, Enable := TRUE, iRepetitionNumber := 0 , iRepetitionPeriod := 0, Comment := '', Param1 := (Set:=0, SetMin:=0, SetMax:=0,Comment:=''), Param2 := (Set:=0, SetMin:=0, SetMax:=0,Comment:='') ),
( sName := 'a_bSafetySLS_GroupError', sClearName := '', sID := '2014', a := FALSE, b := FALSE, iGroup :=2, iSetDelay :=0, iResetDelay := 0, eResetMode := MANU, eBrakeProgram := B1, eAlarmProgram := 0, Enable := TRUE, iRepetitionNumber := 0 , iRepetitionPeriod := 0, Comment := '', Param1 := (Set:=0, SetMin:=0, SetMax:=0,Comment:=''), Param2 := (Set:=0, SetMin:=0, SetMax:=0,Comment:='') ),
( sName := 'a_bSafetyX10_PNOZ_GroupError', sClearName := '', sID := '2015', a := FALSE, b := FALSE, iGroup :=2, iSetDelay :=0, iResetDelay := 0, eResetMode := MANU, eBrakeProgram := B1, eAlarmProgram := 0, Enable := TRUE, iRepetitionNumber := 0 , iRepetitionPeriod := 0, Comment := '', Param1 := (Set:=0, SetMin:=0, SetMax:=0,Comment:=''), Param2 := (Set:=0, SetMin:=0, SetMax:=0,Comment:='') ),
( sName := 'a_bSafetyX6_ExtremFine_GroupError', sClearName := '', sID := '2016', a := FALSE, b := FALSE, iGroup :=2, iSetDelay :=0, iResetDelay := 0, eResetMode := MANU, eBrakeProgram := B1, eAlarmProgram := 0, Enable := TRUE, iRepetitionNumber := 0 , iRepetitionPeriod := 0, Comment := '', Param1 := (Set:=0, SetMin:=0, SetMax:=0,Comment:=''), Param2 := (Set:=0, SetMin:=0, SetMax:=0,Comment:='') ),
( sName := 'a_bSafetyX5_EFC_GroupError', sClearName := '', sID := '2017', a := FALSE, b := FALSE, iGroup :=2, iSetDelay :=0, iResetDelay := 0, eResetMode := MANU, eBrakeProgram := B4, eAlarmProgram := 0, Enable := TRUE, iRepetitionNumber := 0 , iRepetitionPeriod := 0, Comment := '', Param1 := (Set:=0, SetMin:=0, SetMax:=0,Comment:=''), Param2 := (Set:=0, SetMin:=0, SetMax:=0,Comment:='') ),
( sName := 'a_bSafetyFBError', sClearName := '', sID := '2018', a := FALSE, b := FALSE, iGroup :=2, iSetDelay :=0, iResetDelay := 0, eResetMode := MANU, eBrakeProgram := B1, eAlarmProgram := 0, Enable := TRUE, iRepetitionNumber := 0 , iRepetitionPeriod := 0, Comment := '', Param1 := (Set:=0, SetMin:=0, SetMax:=0,Comment:=''), Param2 := (Set:=0, SetMin:=0, SetMax:=0,Comment:='') ),
( sName := 'a_bSafetyCommError', sClearName := '', sID := '2019', a := FALSE, b := FALSE, iGroup :=2, iSetDelay :=0, iResetDelay := 0, eResetMode := MANU, eBrakeProgram := B1, eAlarmProgram := 0, Enable := TRUE, iRepetitionNumber := 0 , iRepetitionPeriod := 0, Comment := '', Param1 := (Set:=0, SetMin:=0, SetMax:=0,Comment:=''), Param2 := (Set:=0, SetMin:=0, SetMax:=0,Comment:='') ),
( sName := 'a_bSafetyOutError', sClearName := '', sID := '2020', a := FALSE, b := FALSE, iGroup :=2, iSetDelay :=0, iResetDelay := 0, eResetMode := MANU, eBrakeProgram := B1, eAlarmProgram := 0, Enable := TRUE, iRepetitionNumber := 0 , iRepetitionPeriod := 0, Comment := '', Param1 := (Set:=0, SetMin:=0, SetMax:=0,Comment:=''), Param2 := (Set:=0, SetMin:=0, SetMax:=0,Comment:='') ),
( sName := 'a_bSafetyOperatorPushButtonEstopTrip', sClearName := '', sID := '2021', a := FALSE, b := FALSE, iGroup :=2, iSetDelay :=0, iResetDelay := 0, eResetMode := MANU, eBrakeProgram := B1, eAlarmProgram := 0, Enable := TRUE, iRepetitionNumber := 0 , iRepetitionPeriod := 0, Comment := '', Param1 := (Set:=0, SetMin:=0, SetMax:=0,Comment:=''), Param2 := (Set:=0, SetMin:=0, SetMax:=0,Comment:='') ),
( sName := 'a_bSafetyHydairSystemEstopTrip', sClearName := '', sID := '2022', a := FALSE, b := FALSE, iGroup :=2, iSetDelay :=0, iResetDelay := 0, eResetMode := MANU, eBrakeProgram := B1, eAlarmProgram := 0, Enable := TRUE, iRepetitionNumber := 0 , iRepetitionPeriod := 0, Comment := '', Param1 := (Set:=0, SetMin:=0, SetMax:=0,Comment:=''), Param2 := (Set:=0, SetMin:=0, SetMax:=0,Comment:='') ),
( sName := 'a_bSafetyPTCSActivatedEstopTrip_ComssLossHydair', sClearName := '', sID := '2023', a := FALSE, b := FALSE, iGroup :=2, iSetDelay :=0, iResetDelay := 0, eResetMode := MANU, eBrakeProgram := B1, eAlarmProgram := 0, Enable := TRUE, iRepetitionNumber := 0 , iRepetitionPeriod := 0, Comment := '', Param1 := (Set:=0, SetMin:=0, SetMax:=0,Comment:=''), Param2 := (Set:=0, SetMin:=0, SetMax:=0,Comment:='') ),
( sName := 'a_bSafetyPTCSActivatedEstopTrip_ExcessiveLoadTestRig', sClearName := '', sID := '2024', a := FALSE, b := FALSE, iGroup :=2, iSetDelay :=0, iResetDelay := 0, eResetMode := MANU, eBrakeProgram := B1, eAlarmProgram := 0, Enable := TRUE, iRepetitionNumber := 0 , iRepetitionPeriod := 0, Comment := '', Param1 := (Set:=0, SetMin:=0, SetMax:=0,Comment:=''), Param2 := (Set:=0, SetMin:=0, SetMax:=0,Comment:='') ),
( sName := 'a_bSafetyPitchSystemEFCActivated', sClearName := '', sID := '2025', a := FALSE, b := FALSE, iGroup :=2, iSetDelay :=0, iResetDelay := 0, eResetMode := MANU, eBrakeProgram := B4, eAlarmProgram := 0, Enable := TRUE, iRepetitionNumber := 0 , iRepetitionPeriod := 0, Comment := '', Param1 := (Set:=0, SetMin:=0, SetMax:=0,Comment:=''), Param2 := (Set:=0, SetMin:=0, SetMax:=0,Comment:='') ),
( sName := 'a_bSafetyEstopResetReq', sClearName := '', sID := '2026', a := FALSE, b := FALSE, iGroup :=2, iSetDelay :=0, iResetDelay := 0, eResetMode := MANU, eBrakeProgram := B99, eAlarmProgram := 0, Enable := TRUE, iRepetitionNumber := 0 , iRepetitionPeriod := 0, Comment := '', Param1 := (Set:=0, SetMin:=0, SetMax:=0,Comment:=''), Param2 := (Set:=0, SetMin:=0, SetMax:=0,Comment:='') ),
( sName := 'a_bSafetyEFCResetReq', sClearName := '', sID := '2027', a := FALSE, b := FALSE, iGroup :=2, iSetDelay :=0, iResetDelay := 0, eResetMode := MANU, eBrakeProgram := B99, eAlarmProgram := 0, Enable := TRUE, iRepetitionNumber := 0 , iRepetitionPeriod := 0, Comment := '', Param1 := (Set:=0, SetMin:=0, SetMax:=0,Comment:=''), Param2 := (Set:=0, SetMin:=0, SetMax:=0,Comment:='') ),
( sName := 'a_bSafetyEstopChainClosed', sClearName := '', sID := '2028', a := FALSE, b := FALSE, iGroup :=2, iSetDelay :=0, iResetDelay := 0, eResetMode := MANU, eBrakeProgram := B99, eAlarmProgram := 0, Enable := TRUE, iRepetitionNumber := 0 , iRepetitionPeriod := 0, Comment := '', Param1 := (Set:=0, SetMin:=0, SetMax:=0,Comment:=''), Param2 := (Set:=0, SetMin:=0, SetMax:=0,Comment:='') ),
( sName := 'a_bSafetyPitchEFCChainClosed', sClearName := '', sID := '2029', a := FALSE, b := FALSE, iGroup :=2, iSetDelay :=0, iResetDelay := 0, eResetMode := MANU, eBrakeProgram := B99, eAlarmProgram := 0, Enable := TRUE, iRepetitionNumber := 0 , iRepetitionPeriod := 0, Comment := '', Param1 := (Set:=0, SetMin:=0, SetMax:=0,Comment:=''), Param2 := (Set:=0, SetMin:=0, SetMax:=0,Comment:='') ),
( sName := 'a_bConverterHeartbeatFailure', sClearName := 'Heartbeat profibus', sID := '3901', a := FALSE, b := FALSE, iGroup :=3, iSetDelay :=10, iResetDelay := 0, eResetMode := MANU, eBrakeProgram := B9, eAlarmProgram := EMAIL, Enable := FALSE, iRepetitionNumber := 0 , iRepetitionPeriod := 10, Comment := 'Heartbeat failed', Param1 := (Set:=0, SetMin:=0, SetMax:=0,Comment:=''), Param2 := (Set:=0, SetMin:=0, SetMax:=0,Comment:='') ),
( sName := 'a_bSSB_NoEFCFromTC', sClearName := 'Water level below slip ring tripped low sensor', sID := '4001', a := FALSE, b := FALSE, iGroup :=4, iSetDelay :=0, iResetDelay := 0, eResetMode := MANU, eBrakeProgram := B4, eAlarmProgram := 0, Enable := TRUE, iRepetitionNumber := 0 , iRepetitionPeriod := 0, Comment := '', Param1 := (Set:=2, SetMin:=1, SetMax:=2,Comment:=''), Param2 := (Set:=0, SetMin:=0, SetMax:=0,Comment:='') ),
( sName := 'a_bSSB_bWatchDogFromPLC', sClearName := 'bWatchDogFromPLC', sID := '4002', a := FALSE, b := FALSE, iGroup :=4, iSetDelay :=0, iResetDelay := 0, eResetMode := MANU, eBrakeProgram := B4, eAlarmProgram := 0, Enable := TRUE, iRepetitionNumber := 0 , iRepetitionPeriod := 0, Comment := '', Param1 := (Set:=0, SetMin:=0, SetMax:=0,Comment:=''), Param2 := (Set:=0, SetMin:=0, SetMax:=0,Comment:='') ),
( sName := 'a_bSSB_bAllBladesAtLimit', sClearName := 'bAllBladesAtLimit', sID := '4003', a := FALSE, b := FALSE, iGroup :=4, iSetDelay :=0, iResetDelay := 0, eResetMode := MANU, eBrakeProgram := B99, eAlarmProgram := 0, Enable := TRUE, iRepetitionNumber := 0 , iRepetitionPeriod := 0, Comment := '', Param1 := (Set:=0, SetMin:=0, SetMax:=0,Comment:=''), Param2 := (Set:=0, SetMin:=0, SetMax:=0,Comment:='') ),
( sName := 'a_bSSB_bAllBladesAtFeather', sClearName := 'bAllBladesAtFeather', sID := '4004', a := FALSE, b := FALSE, iGroup :=4, iSetDelay :=0, iResetDelay := 0, eResetMode := MANU, eBrakeProgram := B99, eAlarmProgram := 0, Enable := TRUE, iRepetitionNumber := 0 , iRepetitionPeriod := 0, Comment := '', Param1 := (Set:=0, SetMin:=0, SetMax:=0,Comment:=''), Param2 := (Set:=0, SetMin:=0, SetMax:=0,Comment:='') ),
( sName := 'a_bSSB_BusOK', sClearName := 'a_bSSB_BusOK', sID := '4005', a := FALSE, b := FALSE, iGroup :=4, iSetDelay :=0, iResetDelay := 0, eResetMode := MANU, eBrakeProgram := B99, eAlarmProgram := 0, Enable := TRUE, iRepetitionNumber := 0 , iRepetitionPeriod := 0, Comment := '', Param1 := (Set:=0, SetMin:=0, SetMax:=0,Comment:=''), Param2 := (Set:=0, SetMin:=0, SetMax:=0,Comment:='') ),
( sName := 'a_bSSB_bCriticalError', sClearName := 'a_bCriticalError', sID := '4006', a := FALSE, b := FALSE, iGroup :=4, iSetDelay :=0, iResetDelay := 0, eResetMode := MANU, eBrakeProgram := B4, eAlarmProgram := 0, Enable := TRUE, iRepetitionNumber := 0 , iRepetitionPeriod := 0, Comment := '', Param1 := (Set:=0, SetMin:=0, SetMax:=0,Comment:=''), Param2 := (Set:=0, SetMin:=0, SetMax:=0,Comment:='') ),
( sName := 'a_bSSB_bFatalError', sClearName := 'a_bFatalError', sID := '4007', a := FALSE, b := FALSE, iGroup :=4, iSetDelay :=0, iResetDelay := 0, eResetMode := MANU, eBrakeProgram := B4, eAlarmProgram := 0, Enable := TRUE, iRepetitionNumber := 0 , iRepetitionPeriod := 0, Comment := '', Param1 := (Set:=0, SetMin:=0, SetMax:=0,Comment:=''), Param2 := (Set:=0, SetMin:=0, SetMax:=0,Comment:='') ),
( sName := 'a_bSSB_bReferencingFailed', sClearName := 'bReferencingFailed', sID := '4008', a := FALSE, b := FALSE, iGroup :=4, iSetDelay :=0, iResetDelay := 0, eResetMode := MANU, eBrakeProgram := B99, eAlarmProgram := 0, Enable := TRUE, iRepetitionNumber := 0 , iRepetitionPeriod := 0, Comment := '', Param1 := (Set:=0, SetMin:=0, SetMax:=0,Comment:=''), Param2 := (Set:=0, SetMin:=0, SetMax:=0,Comment:='') ),
( sName := 'a_bSSB_ExtDI1_Lube1Flt', sClearName := 'a_ExtDI1_Lube1Flt', sID := '4009', a := FALSE, b := FALSE, iGroup :=4, iSetDelay :=0, iResetDelay := 0, eResetMode := MANU, eBrakeProgram := B99, eAlarmProgram := 0, Enable := TRUE, iRepetitionNumber := 0 , iRepetitionPeriod := 0, Comment := '', Param1 := (Set:=0, SetMin:=0, SetMax:=0,Comment:=''), Param2 := (Set:=0, SetMin:=0, SetMax:=0,Comment:='') ),
( sName := 'a_bSSB_PPA_EFC1_by_Error', sClearName := 'a_PPA_EFC1_by_Error', sID := '4010', a := FALSE, b := FALSE, iGroup :=4, iSetDelay :=0, iResetDelay := 0, eResetMode := MANU, eBrakeProgram := B4, eAlarmProgram := 0, Enable := TRUE, iRepetitionNumber := 0 , iRepetitionPeriod := 0, Comment := '', Param1 := (Set:=0, SetMin:=0, SetMax:=0,Comment:=''), Param2 := (Set:=0, SetMin:=0, SetMax:=0,Comment:='') ),
( sName := 'a_bSSB_PPA_EFC1_by_bus', sClearName := 'a_PPA_EFC1_by_bus', sID := '4011', a := FALSE, b := FALSE, iGroup :=4, iSetDelay :=0, iResetDelay := 0, eResetMode := MANU, eBrakeProgram := B4, eAlarmProgram := 0, Enable := TRUE, iRepetitionNumber := 0 , iRepetitionPeriod := 0, Comment := '', Param1 := (Set:=0, SetMin:=0, SetMax:=0,Comment:=''), Param2 := (Set:=0, SetMin:=0, SetMax:=0,Comment:='') ),
( sName := 'a_bSSB_LS_active ', sClearName := 'a_PPA_EFC1_active', sID := '4012', a := FALSE, b := FALSE, iGroup :=4, iSetDelay :=0, iResetDelay := 0, eResetMode := MANU, eBrakeProgram := B99, eAlarmProgram := 0, Enable := TRUE, iRepetitionNumber := 0 , iRepetitionPeriod := 0, Comment := '', Param1 := (Set:=0, SetMin:=0, SetMax:=0,Comment:=''), Param2 := (Set:=0, SetMin:=0, SetMax:=0,Comment:='') ),
( sName := 'a_bSSB_SWLS', sClearName := 'a_bSSB_SWLS', sID := '4013', a := FALSE, b := FALSE, iGroup :=4, iSetDelay :=0, iResetDelay := 0, eResetMode := MANU, eBrakeProgram := B99, eAlarmProgram := 0, Enable := TRUE, iRepetitionNumber := 0 , iRepetitionPeriod := 0, Comment := '', Param1 := (Set:=0, SetMin:=0, SetMax:=0,Comment:=''), Param2 := (Set:=0, SetMin:=0, SetMax:=0,Comment:='') ),
( sName := 'a_bSSB_Bypass1stlimitactive', sClearName := 'a_bSSB_Bypass1stlimitactive', sID := '4014', a := FALSE, b := FALSE, iGroup :=4, iSetDelay :=0, iResetDelay := 0, eResetMode := MANU, eBrakeProgram := B99, eAlarmProgram := 0, Enable := TRUE, iRepetitionNumber := 0 , iRepetitionPeriod := 0, Comment := '', Param1 := (Set:=0, SetMin:=0, SetMax:=0,Comment:=''), Param2 := (Set:=0, SetMin:=0, SetMax:=0,Comment:='') ),
( sName := 'a_bSSB_MainsWarning', sClearName := 'Mains ok (1 = ok, 0 = general warning)', sID := '4015', a := FALSE, b := FALSE, iGroup :=4, iSetDelay :=0, iResetDelay := 0, eResetMode := MANU, eBrakeProgram := B99, eAlarmProgram := 0, Enable := TRUE, iRepetitionNumber := 0 , iRepetitionPeriod := 0, Comment := '', Param1 := (Set:=0, SetMin:=0, SetMax:=0,Comment:=''), Param2 := (Set:=0, SetMin:=0, SetMax:=0,Comment:='') ),
( sName := 'a_bSSB_CurrentBackup_heaterLow', sClearName := 'a_bSSB_CurrentBackup_heaterLow', sID := '4016', a := FALSE, b := FALSE, iGroup :=4, iSetDelay :=0, iResetDelay := 0, eResetMode := MANU, eBrakeProgram := B99, eAlarmProgram := 0, Enable := TRUE, iRepetitionNumber := 0 , iRepetitionPeriod := 0, Comment := '', Param1 := (Set:=0, SetMin:=0, SetMax:=0,Comment:=''), Param2 := (Set:=0, SetMin:=0, SetMax:=0,Comment:='') ),
( sName := 'a_bSSB_Crit_InternEncoderDeviation', sClearName := '; (motor encoder - blade encoder) > uMAX_DEVIATION', sID := '4017', a := FALSE, b := FALSE, iGroup :=4, iSetDelay :=0, iResetDelay := 0, eResetMode := MANU, eBrakeProgram := B4, eAlarmProgram := 0, Enable := TRUE, iRepetitionNumber := 0 , iRepetitionPeriod := 0, Comment := '', Param1 := (Set:=0, SetMin:=0, SetMax:=0,Comment:=''), Param2 := (Set:=0, SetMin:=0, SetMax:=0,Comment:='') ),
( sName := 'a_bSSB_Crit_ExternEncoderDeviation', sClearName := 'a_bSSB_ExternEncoderDeviation', sID := '4018', a := FALSE, b := FALSE, iGroup :=4, iSetDelay :=0, iResetDelay := 0, eResetMode := MANU, eBrakeProgram := B4, eAlarmProgram := 0, Enable := TRUE, iRepetitionNumber := 0 , iRepetitionPeriod := 0, Comment := '', Param1 := (Set:=0, SetMin:=0, SetMax:=0,Comment:=''), Param2 := (Set:=0, SetMin:=0, SetMax:=0,Comment:='') ),
( sName := 'a_bSSB_Backup_Charger_Not_Working', sClearName := '', sID := '4019', a := FALSE, b := FALSE, iGroup :=4, iSetDelay :=0, iResetDelay := 0, eResetMode := MANU, eBrakeProgram := B4, eAlarmProgram := 0, Enable := TRUE, iRepetitionNumber := 0 , iRepetitionPeriod := 0, Comment := '', Param1 := (Set:=0, SetMin:=0, SetMax:=0,Comment:=''), Param2 := (Set:=0, SetMin:=0, SetMax:=0,Comment:='') ),
( sName := 'a_bSSB_Crit_Backup_heating', sClearName := 'a_bSSB_Backup_heating', sID := '4020', a := FALSE, b := FALSE, iGroup :=4, iSetDelay :=0, iResetDelay := 0, eResetMode := MANU, eBrakeProgram := B99, eAlarmProgram := 0, Enable := TRUE, iRepetitionNumber := 0 , iRepetitionPeriod := 0, Comment := '', Param1 := (Set:=0, SetMin:=0, SetMax:=0,Comment:=''), Param2 := (Set:=0, SetMin:=0, SetMax:=0,Comment:='') ),
( sName := 'a_bSSB_Crit_Mains_Not_OK', sClearName := 'a_bSSB_Mains not OK', sID := '4021', a := FALSE, b := FALSE, iGroup :=4, iSetDelay :=0, iResetDelay := 0, eResetMode := MANU, eBrakeProgram := B4, eAlarmProgram := 0, Enable := TRUE, iRepetitionNumber := 0 , iRepetitionPeriod := 0, Comment := '', Param1 := (Set:=0, SetMin:=0, SetMax:=0,Comment:=''), Param2 := (Set:=0, SetMin:=0, SetMax:=0,Comment:='') ),
( sName := 'a_bPPA_ALM_NH', sClearName := '', sID := '4022', a := FALSE, b := FALSE, iGroup :=4, iSetDelay :=0, iResetDelay := 0, eResetMode := MANU, eBrakeProgram := B99, eAlarmProgram := 0, Enable := TRUE, iRepetitionNumber := 0 , iRepetitionPeriod := 0, Comment := 'Error Overspeed', Param1 := (Set:=0, SetMin:=0, SetMax:=0,Comment:=''), Param2 := (Set:=0, SetMin:=0, SetMax:=0,Comment:='') ),
( sName := 'a_bPPA_ALM_UP', sClearName := '', sID := '4023', a := FALSE, b := FALSE, iGroup :=4, iSetDelay :=0, iResetDelay := 0, eResetMode := MANU, eBrakeProgram := B99, eAlarmProgram := 0, Enable := TRUE, iRepetitionNumber := 0 , iRepetitionPeriod := 0, Comment := 'Error Grid(UP)', Param1 := (Set:=0, SetMin:=0, SetMax:=0,Comment:=''), Param2 := (Set:=0, SetMin:=0, SetMax:=0,Comment:='') ),
( sName := 'a_bPPA_ALM_VH', sClearName := '', sID := '4024', a := FALSE, b := FALSE, iGroup :=4, iSetDelay :=0, iResetDelay := 0, eResetMode := MANU, eBrakeProgram := B99, eAlarmProgram := 0, Enable := TRUE, iRepetitionNumber := 0 , iRepetitionPeriod := 0, Comment := 'Error DC Link High', Param1 := (Set:=0, SetMin:=0, SetMax:=0,Comment:=''), Param2 := (Set:=0, SetMin:=0, SetMax:=0,Comment:='') ),
( sName := 'a_bPPA_ALM_VL', sClearName := '', sID := '4025', a := FALSE, b := FALSE, iGroup :=4, iSetDelay :=0, iResetDelay := 0, eResetMode := MANU, eBrakeProgram := B99, eAlarmProgram := 0, Enable := TRUE, iRepetitionNumber := 0 , iRepetitionPeriod := 0, Comment := 'Error DC Link Low', Param1 := (Set:=0, SetMin:=0, SetMax:=0,Comment:=''), Param2 := (Set:=0, SetMin:=0, SetMax:=0,Comment:='') ),
( sName := 'a_bPPA_ALM_VU', sClearName := '', sID := '4026', a := FALSE, b := FALSE, iGroup :=4, iSetDelay :=0, iResetDelay := 0, eResetMode := MANU, eBrakeProgram := B99, eAlarmProgram := 0, Enable := TRUE, iRepetitionNumber := 0 , iRepetitionPeriod := 0, Comment := 'Error DC Link unplausable', Param1 := (Set:=0, SetMin:=0, SetMax:=0,Comment:=''), Param2 := (Set:=0, SetMin:=0, SetMax:=0,Comment:='') ),
( sName := 'a_bPPA_ALM_OO', sClearName := '', sID := '4027', a := FALSE, b := FALSE, iGroup :=4, iSetDelay :=0, iResetDelay := 0, eResetMode := MANU, eBrakeProgram := B99, eAlarmProgram := 0, Enable := TRUE, iRepetitionNumber := 0 , iRepetitionPeriod := 0, Comment := 'Error Open Output', Param1 := (Set:=0, SetMin:=0, SetMax:=0,Comment:=''), Param2 := (Set:=0, SetMin:=0, SetMax:=0,Comment:='') ),
( sName := 'a_bPPA_ALM_RB', sClearName := '', sID := '4028', a := FALSE, b := FALSE, iGroup :=4, iSetDelay :=0, iResetDelay := 0, eResetMode := MANU, eBrakeProgram := B99, eAlarmProgram := 0, Enable := TRUE, iRepetitionNumber := 0 , iRepetitionPeriod := 0, Comment := 'Error Brake Chopper', Param1 := (Set:=0, SetMin:=0, SetMax:=0,Comment:=''), Param2 := (Set:=0, SetMin:=0, SetMax:=0,Comment:='') ),
( sName := 'a_bPPA_ALM_OF', sClearName := '', sID := '4029', a := FALSE, b := FALSE, iGroup :=4, iSetDelay :=0, iResetDelay := 0, eResetMode := MANU, eBrakeProgram := B99, eAlarmProgram := 0, Enable := TRUE, iRepetitionNumber := 0 , iRepetitionPeriod := 0, Comment := 'Error Overload IGBT', Param1 := (Set:=0, SetMin:=0, SetMax:=0,Comment:=''), Param2 := (Set:=0, SetMin:=0, SetMax:=0,Comment:='') ),
( sName := 'a_bPPA_ALM_OC', sClearName := '', sID := '4030', a := FALSE, b := FALSE, iGroup :=4, iSetDelay :=0, iResetDelay := 0, eResetMode := MANU, eBrakeProgram := B99, eAlarmProgram := 0, Enable := TRUE, iRepetitionNumber := 0 , iRepetitionPeriod := 0, Comment := 'Error Overcurrent', Param1 := (Set:=0, SetMin:=0, SetMax:=0,Comment:=''), Param2 := (Set:=0, SetMin:=0, SetMax:=0,Comment:='') ),
( sName := 'a_bPPA_ALM_CF', sClearName := '', sID := '4031', a := FALSE, b := FALSE, iGroup :=4, iSetDelay :=0, iResetDelay := 0, eResetMode := MANU, eBrakeProgram := B99, eAlarmProgram := 0, Enable := TRUE, iRepetitionNumber := 0 , iRepetitionPeriod := 0, Comment := 'Error Current -V', Param1 := (Set:=0, SetMin:=0, SetMax:=0,Comment:=''), Param2 := (Set:=0, SetMin:=0, SetMax:=0,Comment:='') ),
( sName := 'a_bPPA_ALM_IS', sClearName := '', sID := '4032', a := FALSE, b := FALSE, iGroup :=4, iSetDelay :=0, iResetDelay := 0, eResetMode := MANU, eBrakeProgram := B99, eAlarmProgram := 0, Enable := TRUE, iRepetitionNumber := 0 , iRepetitionPeriod := 0, Comment := 'Error Internal Supply', Param1 := (Set:=0, SetMin:=0, SetMax:=0,Comment:=''), Param2 := (Set:=0, SetMin:=0, SetMax:=0,Comment:='') ),
( sName := 'a_bPPA_ALM_VE', sClearName := '', sID := '4033', a := FALSE, b := FALSE, iGroup :=4, iSetDelay :=0, iResetDelay := 0, eResetMode := MANU, eBrakeProgram := B99, eAlarmProgram := 0, Enable := TRUE, iRepetitionNumber := 0 , iRepetitionPeriod := 0, Comment := 'Error Electronic supply', Param1 := (Set:=0, SetMin:=0, SetMax:=0,Comment:=''), Param2 := (Set:=0, SetMin:=0, SetMax:=0,Comment:='') ),
( sName := 'a_bPPA_ALM_HF', sClearName := '', sID := '4034', a := FALSE, b := FALSE, iGroup :=4, iSetDelay :=0, iResetDelay := 0, eResetMode := MANU, eBrakeProgram := B99, eAlarmProgram := 0, Enable := TRUE, iRepetitionNumber := 0 , iRepetitionPeriod := 0, Comment := 'Error Hardware Failure', Param1 := (Set:=0, SetMin:=0, SetMax:=0,Comment:=''), Param2 := (Set:=0, SetMin:=0, SetMax:=0,Comment:='') ),
( sName := 'a_bPPA_ALM_PE', sClearName := '', sID := '4035', a := FALSE, b := FALSE, iGroup :=4, iSetDelay :=0, iResetDelay := 0, eResetMode := MANU, eBrakeProgram := B99, eAlarmProgram := 0, Enable := TRUE, iRepetitionNumber := 0 , iRepetitionPeriod := 0, Comment := 'Error Parameter Loading', Param1 := (Set:=0, SetMin:=0, SetMax:=0,Comment:=''), Param2 := (Set:=0, SetMin:=0, SetMax:=0,Comment:='') ),
( sName := 'a_bPPA_ALM_MM', sClearName := '', sID := '4036', a := FALSE, b := FALSE, iGroup :=4, iSetDelay :=0, iResetDelay := 0, eResetMode := MANU, eBrakeProgram := B99, eAlarmProgram := 0, Enable := TRUE, iRepetitionNumber := 0 , iRepetitionPeriod := 0, Comment := 'Error Motor lxt', Param1 := (Set:=0, SetMin:=0, SetMax:=0,Comment:=''), Param2 := (Set:=0, SetMin:=0, SetMax:=0,Comment:='') ),
( sName := 'a_bPPA_ALM_CP', sClearName := '', sID := '4037', a := FALSE, b := FALSE, iGroup :=4, iSetDelay :=0, iResetDelay := 0, eResetMode := MANU, eBrakeProgram := B99, eAlarmProgram := 0, Enable := TRUE, iRepetitionNumber := 0 , iRepetitionPeriod := 0, Comment := 'Error Preogram', Param1 := (Set:=0, SetMin:=0, SetMax:=0,Comment:=''), Param2 := (Set:=0, SetMin:=0, SetMax:=0,Comment:='') ),
( sName := 'a_bPPA_ALM_EE', sClearName := '', sID := '4038', a := FALSE, b := FALSE, iGroup :=4, iSetDelay :=0, iResetDelay := 0, eResetMode := MANU, eBrakeProgram := B99, eAlarmProgram := 0, Enable := TRUE, iRepetitionNumber := 0 , iRepetitionPeriod := 0, Comment := 'Error EEPROM', Param1 := (Set:=0, SetMin:=0, SetMax:=0,Comment:=''), Param2 := (Set:=0, SetMin:=0, SetMax:=0,Comment:='') ),
( sName := 'a_bPPA_ALM_SB', sClearName := '', sID := '4039', a := FALSE, b := FALSE, iGroup :=4, iSetDelay :=0, iResetDelay := 0, eResetMode := MANU, eBrakeProgram := B99, eAlarmProgram := 0, Enable := TRUE, iRepetitionNumber := 0 , iRepetitionPeriod := 0, Comment := 'Error SSB Bus', Param1 := (Set:=0, SetMin:=0, SetMax:=0,Comment:=''), Param2 := (Set:=0, SetMin:=0, SetMax:=0,Comment:='') ),
( sName := 'a_bPPA_ALM_E1', sClearName := '', sID := '4040', a := FALSE, b := FALSE, iGroup :=4, iSetDelay :=0, iResetDelay := 0, eResetMode := MANU, eBrakeProgram := B99, eAlarmProgram := 0, Enable := TRUE, iRepetitionNumber := 0 , iRepetitionPeriod := 0, Comment := 'Error Encoder 1', Param1 := (Set:=0, SetMin:=0, SetMax:=0,Comment:=''), Param2 := (Set:=0, SetMin:=0, SetMax:=0,Comment:='') ),
( sName := 'a_bPPA_ALM_E2', sClearName := '', sID := '4041', a := FALSE, b := FALSE, iGroup :=4, iSetDelay :=0, iResetDelay := 0, eResetMode := MANU, eBrakeProgram := B99, eAlarmProgram := 0, Enable := TRUE, iRepetitionNumber := 0 , iRepetitionPeriod := 0, Comment := 'Error Encoder 2', Param1 := (Set:=0, SetMin:=0, SetMax:=0,Comment:=''), Param2 := (Set:=0, SetMin:=0, SetMax:=0,Comment:='') ),
( sName := 'a_bPPA_ALM_SL', sClearName := '', sID := '4042', a := FALSE, b := FALSE, iGroup :=4, iSetDelay :=0, iResetDelay := 0, eResetMode := MANU, eBrakeProgram := B99, eAlarmProgram := 0, Enable := TRUE, iRepetitionNumber := 0 , iRepetitionPeriod := 0, Comment := 'Error SWLS', Param1 := (Set:=0, SetMin:=0, SetMax:=0,Comment:=''), Param2 := (Set:=0, SetMin:=0, SetMax:=0,Comment:='') ),
( sName := 'a_bPPA_ALM_SF', sClearName := '', sID := '4043', a := FALSE, b := FALSE, iGroup :=4, iSetDelay :=0, iResetDelay := 0, eResetMode := MANU, eBrakeProgram := B99, eAlarmProgram := 0, Enable := TRUE, iRepetitionNumber := 0 , iRepetitionPeriod := 0, Comment := 'Error Speed Feedback', Param1 := (Set:=0, SetMin:=0, SetMax:=0,Comment:=''), Param2 := (Set:=0, SetMin:=0, SetMax:=0,Comment:='') ),
( sName := 'a_bPPA_ALM_PF', sClearName := '', sID := '4044', a := FALSE, b := FALSE, iGroup :=4, iSetDelay :=0, iResetDelay := 0, eResetMode := MANU, eBrakeProgram := B99, eAlarmProgram := 0, Enable := TRUE, iRepetitionNumber := 0 , iRepetitionPeriod := 0, Comment := 'Error Position', Param1 := (Set:=0, SetMin:=0, SetMax:=0,Comment:=''), Param2 := (Set:=0, SetMin:=0, SetMax:=0,Comment:='') ),
( sName := 'a_bPPA_ALM_BH', sClearName := '', sID := '4045', a := FALSE, b := FALSE, iGroup :=4, iSetDelay :=0, iResetDelay := 0, eResetMode := MANU, eBrakeProgram := B99, eAlarmProgram := 0, Enable := TRUE, iRepetitionNumber := 0 , iRepetitionPeriod := 0, Comment := 'Error Brake Current High', Param1 := (Set:=0, SetMin:=0, SetMax:=0,Comment:=''), Param2 := (Set:=0, SetMin:=0, SetMax:=0,Comment:='') ),
( sName := 'a_bPPA_ALM_BL', sClearName := '', sID := '4046', a := FALSE, b := FALSE, iGroup :=4, iSetDelay :=0, iResetDelay := 0, eResetMode := MANU, eBrakeProgram := B99, eAlarmProgram := 0, Enable := TRUE, iRepetitionNumber := 0 , iRepetitionPeriod := 0, Comment := 'Error Brake Current Low', Param1 := (Set:=0, SetMin:=0, SetMax:=0,Comment:=''), Param2 := (Set:=0, SetMin:=0, SetMax:=0,Comment:='') ),
( sName := 'a_bPPA_ALM_BD', sClearName := '', sID := '4047', a := FALSE, b := FALSE, iGroup :=4, iSetDelay :=0, iResetDelay := 0, eResetMode := MANU, eBrakeProgram := B99, eAlarmProgram := 0, Enable := TRUE, iRepetitionNumber := 0 , iRepetitionPeriod := 0, Comment := 'Error Brake Drive', Param1 := (Set:=0, SetMin:=0, SetMax:=0,Comment:=''), Param2 := (Set:=0, SetMin:=0, SetMax:=0,Comment:='') ),
( sName := 'a_bPPA_ALM_MT', sClearName := '', sID := '4048', a := FALSE, b := FALSE, iGroup :=4, iSetDelay :=0, iResetDelay := 0, eResetMode := MANU, eBrakeProgram := B99, eAlarmProgram := 0, Enable := TRUE, iRepetitionNumber := 0 , iRepetitionPeriod := 0, Comment := 'Error Motor Temperature', Param1 := (Set:=0, SetMin:=0, SetMax:=0,Comment:=''), Param2 := (Set:=0, SetMin:=0, SetMax:=0,Comment:='') ),
( sName := 'a_bPPA_ALM_HT', sClearName := '', sID := '4049', a := FALSE, b := FALSE, iGroup :=4, iSetDelay :=0, iResetDelay := 0, eResetMode := MANU, eBrakeProgram := B99, eAlarmProgram := 0, Enable := TRUE, iRepetitionNumber := 0 , iRepetitionPeriod := 0, Comment := 'Error Heat Sink Temp', Param1 := (Set:=0, SetMin:=0, SetMax:=0,Comment:=''), Param2 := (Set:=0, SetMin:=0, SetMax:=0,Comment:='') ),
( sName := 'a_bPPA_ALM_TL', sClearName := '', sID := '4050', a := FALSE, b := FALSE, iGroup :=4, iSetDelay :=0, iResetDelay := 0, eResetMode := MANU, eBrakeProgram := B99, eAlarmProgram := 0, Enable := TRUE, iRepetitionNumber := 0 , iRepetitionPeriod := 0, Comment := 'Error Control board Temp Low', Param1 := (Set:=0, SetMin:=0, SetMax:=0,Comment:=''), Param2 := (Set:=0, SetMin:=0, SetMax:=0,Comment:='') ),
( sName := 'a_bPPA_ALM_T1', sClearName := '', sID := '4051', a := FALSE, b := FALSE, iGroup :=4, iSetDelay :=0, iResetDelay := 0, eResetMode := MANU, eBrakeProgram := B99, eAlarmProgram := 0, Enable := TRUE, iRepetitionNumber := 0 , iRepetitionPeriod := 0, Comment := 'Error Control board temp High', Param1 := (Set:=0, SetMin:=0, SetMax:=0,Comment:=''), Param2 := (Set:=0, SetMin:=0, SetMax:=0,Comment:='') ),
( sName := 'a_bPPA_ALM_T2', sClearName := '', sID := '4052', a := FALSE, b := FALSE, iGroup :=4, iSetDelay :=0, iResetDelay := 0, eResetMode := MANU, eBrakeProgram := B99, eAlarmProgram := 0, Enable := TRUE, iRepetitionNumber := 0 , iRepetitionPeriod := 0, Comment := 'Error Power supply temp', Param1 := (Set:=0, SetMin:=0, SetMax:=0,Comment:=''), Param2 := (Set:=0, SetMin:=0, SetMax:=0,Comment:='') ),
( sName := 'a_bPPA_ALM_CR', sClearName := '', sID := '4053', a := FALSE, b := FALSE, iGroup :=4, iSetDelay :=0, iResetDelay := 0, eResetMode := MANU, eBrakeProgram := B99, eAlarmProgram := 0, Enable := TRUE, iRepetitionNumber := 0 , iRepetitionPeriod := 0, Comment := 'Error Controlled Rectifier', Param1 := (Set:=0, SetMin:=0, SetMax:=0,Comment:=''), Param2 := (Set:=0, SetMin:=0, SetMax:=0,Comment:='') ),
( sName := 'a_bPPA_ALM_TT', sClearName := '', sID := '4054', a := FALSE, b := FALSE, iGroup :=4, iSetDelay :=0, iResetDelay := 0, eResetMode := MANU, eBrakeProgram := B99, eAlarmProgram := 0, Enable := TRUE, iRepetitionNumber := 0 , iRepetitionPeriod := 0, Comment := 'Error IGBT Temp', Param1 := (Set:=0, SetMin:=0, SetMax:=0,Comment:=''), Param2 := (Set:=0, SetMin:=0, SetMax:=0,Comment:='') ),
( sName := 'a_bPPA_ALM_S1', sClearName := '', sID := '4055', a := FALSE, b := FALSE, iGroup :=4, iSetDelay :=0, iResetDelay := 0, eResetMode := MANU, eBrakeProgram := B99, eAlarmProgram := 0, Enable := TRUE, iRepetitionNumber := 0 , iRepetitionPeriod := 0, Comment := 'Error ICO Slave 1', Param1 := (Set:=0, SetMin:=0, SetMax:=0,Comment:=''), Param2 := (Set:=0, SetMin:=0, SetMax:=0,Comment:='') ),
( sName := 'a_bPPA_ALM_S2', sClearName := '', sID := '4056', a := FALSE, b := FALSE, iGroup :=4, iSetDelay :=0, iResetDelay := 0, eResetMode := MANU, eBrakeProgram := B99, eAlarmProgram := 0, Enable := TRUE, iRepetitionNumber := 0 , iRepetitionPeriod := 0, Comment := 'Error ICO Slave 2', Param1 := (Set:=0, SetMin:=0, SetMax:=0,Comment:=''), Param2 := (Set:=0, SetMin:=0, SetMax:=0,Comment:='') ),
( sName := 'a_bPPA_ALM_HB', sClearName := '', sID := '4057', a := FALSE, b := FALSE, iGroup :=4, iSetDelay :=0, iResetDelay := 0, eResetMode := MANU, eBrakeProgram := B99, eAlarmProgram := 0, Enable := TRUE, iRepetitionNumber := 0 , iRepetitionPeriod := 0, Comment := 'Error Back up voltage high', Param1 := (Set:=0, SetMin:=0, SetMax:=0,Comment:=''), Param2 := (Set:=0, SetMin:=0, SetMax:=0,Comment:='') ),
( sName := 'a_bPPA_ALM_LB', sClearName := '', sID := '4058', a := FALSE, b := FALSE, iGroup :=4, iSetDelay :=0, iResetDelay := 0, eResetMode := MANU, eBrakeProgram := B99, eAlarmProgram := 0, Enable := TRUE, iRepetitionNumber := 0 , iRepetitionPeriod := 0, Comment := 'Error Back up voltage Low', Param1 := (Set:=0, SetMin:=0, SetMax:=0,Comment:=''), Param2 := (Set:=0, SetMin:=0, SetMax:=0,Comment:='') ),
( sName := 'a_bPPA_ALM_RS', sClearName := '', sID := '4059', a := FALSE, b := FALSE, iGroup :=4, iSetDelay :=0, iResetDelay := 0, eResetMode := MANU, eBrakeProgram := B99, eAlarmProgram := 0, Enable := TRUE, iRepetitionNumber := 0 , iRepetitionPeriod := 0, Comment := 'Error Resolver sync', Param1 := (Set:=0, SetMin:=0, SetMax:=0,Comment:=''), Param2 := (Set:=0, SetMin:=0, SetMax:=0,Comment:='') ),
( sName := 'a_bPPA_ALM_RR', sClearName := '', sID := '4060', a := FALSE, b := FALSE, iGroup :=4, iSetDelay :=0, iResetDelay := 0, eResetMode := MANU, eBrakeProgram := B99, eAlarmProgram := 0, Enable := TRUE, iRepetitionNumber := 0 , iRepetitionPeriod := 0, Comment := 'Error Resolver Reference', Param1 := (Set:=0, SetMin:=0, SetMax:=0,Comment:=''), Param2 := (Set:=0, SetMin:=0, SetMax:=0,Comment:='') ),
( sName := 'a_bPPA_ALM_CE', sClearName := '', sID := '4061', a := FALSE, b := FALSE, iGroup :=4, iSetDelay :=0, iResetDelay := 0, eResetMode := MANU, eBrakeProgram := B99, eAlarmProgram := 0, Enable := TRUE, iRepetitionNumber := 0 , iRepetitionPeriod := 0, Comment := 'Error CANext', Param1 := (Set:=0, SetMin:=0, SetMax:=0,Comment:=''), Param2 := (Set:=0, SetMin:=0, SetMax:=0,Comment:='') ),
( sName := 'a_bPPA_ALM_C2', sClearName := '', sID := '4062', a := FALSE, b := FALSE, iGroup :=4, iSetDelay :=0, iResetDelay := 0, eResetMode := MANU, eBrakeProgram := B99, eAlarmProgram := 0, Enable := TRUE, iRepetitionNumber := 0 , iRepetitionPeriod := 0, Comment := 'Error ', Param1 := (Set:=0, SetMin:=0, SetMax:=0,Comment:=''), Param2 := (Set:=0, SetMin:=0, SetMax:=0,Comment:='') ),
( sName := 'a_bPPA_ALM_PS', sClearName := '', sID := '4063', a := FALSE, b := FALSE, iGroup :=4, iSetDelay :=0, iResetDelay := 0, eResetMode := MANU, eBrakeProgram := B99, eAlarmProgram := 0, Enable := TRUE, iRepetitionNumber := 0 , iRepetitionPeriod := 0, Comment := 'Error ', Param1 := (Set:=0, SetMin:=0, SetMax:=0,Comment:=''), Param2 := (Set:=0, SetMin:=0, SetMax:=0,Comment:='') ),
( sName := 'a_bPPA_ALM_QC', sClearName := '', sID := '4064', a := FALSE, b := FALSE, iGroup :=4, iSetDelay :=0, iResetDelay := 0, eResetMode := MANU, eBrakeProgram := B99, eAlarmProgram := 0, Enable := TRUE, iRepetitionNumber := 0 , iRepetitionPeriod := 0, Comment := 'Error ', Param1 := (Set:=0, SetMin:=0, SetMax:=0,Comment:=''), Param2 := (Set:=0, SetMin:=0, SetMax:=0,Comment:='') ),
( sName := 'a_bPPA_ALM_RE', sClearName := '', sID := '4065', a := FALSE, b := FALSE, iGroup :=4, iSetDelay :=0, iResetDelay := 0, eResetMode := MANU, eBrakeProgram := B99, eAlarmProgram := 0, Enable := TRUE, iRepetitionNumber := 0 , iRepetitionPeriod := 0, Comment := 'Error Value Range Extended', Param1 := (Set:=0, SetMin:=0, SetMax:=0,Comment:=''), Param2 := (Set:=0, SetMin:=0, SetMax:=0,Comment:='') ),
( sName := 'a_bNoSSBBusFailureANDAllSlavesStatusOnline', sClearName := '', sID := '4066', a := FALSE, b := FALSE, iGroup :=4, iSetDelay :=0, iResetDelay := 0, eResetMode := MANU, eBrakeProgram := B99, eAlarmProgram := 0, Enable := TRUE, iRepetitionNumber := 0 , iRepetitionPeriod := 0, Comment := '', Param1 := (Set:=0, SetMin:=0, SetMax:=0,Comment:=''), Param2 := (Set:=0, SetMin:=0, SetMax:=0,Comment:='') ),
( sName := 'a_bNoCommunicationTOANYSlave', sClearName := '', sID := '4067', a := FALSE, b := FALSE, iGroup :=4, iSetDelay :=0, iResetDelay := 0, eResetMode := MANU, eBrakeProgram := B99, eAlarmProgram := 0, Enable := TRUE, iRepetitionNumber := 0 , iRepetitionPeriod := 0, Comment := 'System Fatal Error bit 4 SSB to any slave not ok', Param1 := (Set:=0, SetMin:=0, SetMax:=0,Comment:=''), Param2 := (Set:=0, SetMin:=0, SetMax:=0,Comment:='') ),
( sName := 'a_bSSB_NoCommunicationTOPLCMaster', sClearName := '', sID := '4068', a := FALSE, b := FALSE, iGroup :=4, iSetDelay :=0, iResetDelay := 0, eResetMode := MANU, eBrakeProgram := B99, eAlarmProgram := 0, Enable := TRUE, iRepetitionNumber := 0 , iRepetitionPeriod := 0, Comment := '', Param1 := (Set:=0, SetMin:=0, SetMax:=0,Comment:=''), Param2 := (Set:=0, SetMin:=0, SetMax:=0,Comment:='') ),
( sName := 'a_bSSB_NoCommunicationTOSlave1_SCI', sClearName := '', sID := '4069', a := FALSE, b := FALSE, iGroup :=4, iSetDelay :=0, iResetDelay := 0, eResetMode := MANU, eBrakeProgram := B99, eAlarmProgram := 0, Enable := TRUE, iRepetitionNumber := 0 , iRepetitionPeriod := 0, Comment := '', Param1 := (Set:=0, SetMin:=0, SetMax:=0,Comment:=''), Param2 := (Set:=0, SetMin:=0, SetMax:=0,Comment:='') ),
( sName := 'a_bSSB_NoCommunicationTOSlave2_PPAM1', sClearName := '', sID := '4070', a := FALSE, b := FALSE, iGroup :=4, iSetDelay :=0, iResetDelay := 0, eResetMode := MANU, eBrakeProgram := B99, eAlarmProgram := 0, Enable := TRUE, iRepetitionNumber := 0 , iRepetitionPeriod := 0, Comment := '', Param1 := (Set:=0, SetMin:=0, SetMax:=0,Comment:=''), Param2 := (Set:=0, SetMin:=0, SetMax:=0,Comment:='') ),
( sName := 'a_bSSB_NoCommunicationTOSlave3_PPAM2', sClearName := '', sID := '4071', a := FALSE, b := FALSE, iGroup :=4, iSetDelay :=0, iResetDelay := 0, eResetMode := MANU, eBrakeProgram := B99, eAlarmProgram := 0, Enable := TRUE, iRepetitionNumber := 0 , iRepetitionPeriod := 0, Comment := '', Param1 := (Set:=0, SetMin:=0, SetMax:=0,Comment:=''), Param2 := (Set:=0, SetMin:=0, SetMax:=0,Comment:='') ),
( sName := 'a_bSSB_NoCommunicationTOSlave4_PPAM3', sClearName := '', sID := '4072', a := FALSE, b := FALSE, iGroup :=4, iSetDelay :=0, iResetDelay := 0, eResetMode := MANU, eBrakeProgram := B99, eAlarmProgram := 0, Enable := TRUE, iRepetitionNumber := 0 , iRepetitionPeriod := 0, Comment := '', Param1 := (Set:=0, SetMin:=0, SetMax:=0,Comment:=''), Param2 := (Set:=0, SetMin:=0, SetMax:=0,Comment:='') ),
( sName := 'a_bSSB_NoCommunicationToPLCFromSlave2PPAMaster1', sClearName := '', sID := '4073', a := FALSE, b := FALSE, iGroup :=4, iSetDelay :=0, iResetDelay := 0, eResetMode := MANU, eBrakeProgram := B99, eAlarmProgram := 0, Enable := TRUE, iRepetitionNumber := 0 , iRepetitionPeriod := 0, Comment := 'system fatal Slave 2 PPA2 not ok', Param1 := (Set:=0, SetMin:=0, SetMax:=0,Comment:=''), Param2 := (Set:=0, SetMin:=0, SetMax:=0,Comment:='') ),
( sName := 'a_bSSB_NoCommunicationToPLCFromSlave3PPAMaster2', sClearName := '', sID := '4074', a := FALSE, b := FALSE, iGroup :=4, iSetDelay :=0, iResetDelay := 0, eResetMode := MANU, eBrakeProgram := B99, eAlarmProgram := 0, Enable := TRUE, iRepetitionNumber := 0 , iRepetitionPeriod := 0, Comment := '', Param1 := (Set:=0, SetMin:=0, SetMax:=0,Comment:=''), Param2 := (Set:=0, SetMin:=0, SetMax:=0,Comment:='') ),
( sName := 'a_bSSB_NoCommunicationToPLCFromSlave4PPAMaster3', sClearName := '', sID := '4075', a := FALSE, b := FALSE, iGroup :=4, iSetDelay :=0, iResetDelay := 0, eResetMode := MANU, eBrakeProgram := B99, eAlarmProgram := 0, Enable := TRUE, iRepetitionNumber := 0 , iRepetitionPeriod := 0, Comment := '', Param1 := (Set:=0, SetMin:=0, SetMax:=0,Comment:=''), Param2 := (Set:=0, SetMin:=0, SetMax:=0,Comment:='') ),
( sName := 'a_bSSB_NotReadyToOperate', sClearName := '', sID := '4076', a := FALSE, b := FALSE, iGroup :=4, iSetDelay :=0, iResetDelay := 0, eResetMode := MANU, eBrakeProgram := B99, eAlarmProgram := 0, Enable := TRUE, iRepetitionNumber := 0 , iRepetitionPeriod := 0, Comment := '', Param1 := (Set:=0, SetMin:=0, SetMax:=0,Comment:=''), Param2 := (Set:=0, SetMin:=0, SetMax:=0,Comment:='') ),
( sName := 'a_bPitchEncodersDisagreeSSB_Safety', sClearName := 'Encoders readings differ with SSB derived blade measurements above acceptable thresholds', sID := '4062', a := FALSE, b := FALSE, iGroup :=4, iSetDelay :=1, iResetDelay := 1, eResetMode := MANU, eBrakeProgram := B4, eAlarmProgram := 0, Enable := TRUE, iRepetitionNumber := 0 , iRepetitionPeriod := 0, Comment := 'Encoders readings differ with SSB derived blade measurements more than acceptable thresholds. Trip safety circuit.', Param1 := (Set:=3, SetMin:=3, SetMax:=3,Comment:='Degs'), Param2 := (Set:=1, SetMin:=1, SetMax:=1,Comment:='Degs') ),
( sName := 'a_bPitchEncodersDisagreeSSB_Fault', sClearName := 'Encoders readings differ with SSB derived blade measurements above acceptable thresholds', sID := '4063', a := FALSE, b := FALSE, iGroup :=4, iSetDelay :=1, iResetDelay := 1, eResetMode := MANU, eBrakeProgram := B20, eAlarmProgram := 0, Enable := TRUE, iRepetitionNumber := 0 , iRepetitionPeriod := 0, Comment := 'Encoders readings differ with SSB derived blade measurements more than acceptable thresholds. Initiate controlled shutdown.', Param1 := (Set:=1.99999971123577, SetMin:=1.99999971123577, SetMax:=1.99999971123577,Comment:='Degs'), Param2 := (Set:=1, SetMin:=1, SetMax:=1,Comment:='Degs') ),
( sName := 'a_bPitchEncodersDisagreeSSB_Warning', sClearName := 'Encoders readings differ with SSB derived blade measurements above acceptable thresholds', sID := '4064', a := FALSE, b := FALSE, iGroup :=4, iSetDelay :=1, iResetDelay := 1, eResetMode := MANU, eBrakeProgram := B99, eAlarmProgram := 0, Enable := TRUE, iRepetitionNumber := 0 , iRepetitionPeriod := 0, Comment := 'Encoders readings differ with SSB derived blade measurements more than acceptable thresholds. Notify operator', Param1 := (Set:=1.5, SetMin:=1.5, SetMax:=1.5,Comment:='Degs'), Param2 := (Set:=1, SetMin:=1, SetMax:=1,Comment:='Degs') ),
( sName := 'a_bPitchTorqueAv1sHiWarn', sClearName := 'Higher than normal torque spikes on active SSB drive warning', sID := '4080', a := FALSE, b := FALSE, iGroup :=4, iSetDelay :=1, iResetDelay := 1, eResetMode := MANU, eBrakeProgram := B99, eAlarmProgram := 0, Enable := TRUE, iRepetitionNumber := 0 , iRepetitionPeriod := 0, Comment := 'Higher than normal torque spikes on active SSB drive warning', Param1 := (Set:=300, SetMin:=0, SetMax:=320,Comment:=''), Param2 := (Set:=100, SetMin:=0, SetMax:=100,Comment:='') ),
( sName := 'a_bPitchTorqueAv1sHiAlarm', sClearName := 'Higher than normal torque spikes on active SSB drive alarm', sID := '4081', a := FALSE, b := FALSE, iGroup :=4, iSetDelay :=1, iResetDelay := 1, eResetMode := MANU, eBrakeProgram := B20, eAlarmProgram := 0, Enable := TRUE, iRepetitionNumber := 0 , iRepetitionPeriod := 0, Comment := 'Higher than normal torque spikes on active SSB drive alarm', Param1 := (Set:=320, SetMin:=0, SetMax:=320,Comment:=''), Param2 := (Set:=100, SetMin:=0, SetMax:=100,Comment:='') ),
( sName := 'a_bPitchTorqueAv5sTorqueHiWarn', sClearName := 'Higher than normal steady state torques on active SSB drive warning', sID := '4082', a := FALSE, b := FALSE, iGroup :=4, iSetDelay :=1, iResetDelay := 1, eResetMode := MANU, eBrakeProgram := B99, eAlarmProgram := 0, Enable := TRUE, iRepetitionNumber := 0 , iRepetitionPeriod := 0, Comment := 'Higher than normal steady state torques on active SSB drive', Param1 := (Set:=320, SetMin:=0, SetMax:=320,Comment:=''), Param2 := (Set:=100, SetMin:=0, SetMax:=100,Comment:='') ),
( sName := 'a_bPitchTorqueAv60sTorqueHiWarn', sClearName := 'Higher than normal average torque levels seen on SSB system warning', sID := '4083', a := FALSE, b := FALSE, iGroup :=4, iSetDelay :=1, iResetDelay := 1, eResetMode := MANU, eBrakeProgram := B99, eAlarmProgram := 0, Enable := TRUE, iRepetitionNumber := 0 , iRepetitionPeriod := 0, Comment := 'Higher than normal average torque levels seen on SSB system', Param1 := (Set:=320, SetMin:=0, SetMax:=320,Comment:=''), Param2 := (Set:=100, SetMin:=0, SetMax:=100,Comment:='') ),
( sName := 'a_bPitchDiffInStopPos', sClearName := 'Difference in pitch and feather STOP position. ', sID := '4084', a := FALSE, b := FALSE, iGroup :=4, iSetDelay :=1, iResetDelay := 1, eResetMode := MANU, eBrakeProgram := B99, eAlarmProgram := 0, Enable := TRUE, iRepetitionNumber := 0 , iRepetitionPeriod := 0, Comment := 'Difference in pitch and feather STOP position. ', Param1 := (Set:=0.4, SetMin:=0, SetMax:=2,Comment:=''), Param2 := (Set:=0.2, SetMin:=0, SetMax:=0.2,Comment:='') ),
( sName := 'a_bPitchMaxMotorTorqueExceeded', sClearName := 'Pitch Max motor torque exceeded', sID := '4085', a := FALSE, b := FALSE, iGroup :=4, iSetDelay :=1, iResetDelay := 1, eResetMode := MANU, eBrakeProgram := B20, eAlarmProgram := 0, Enable := TRUE, iRepetitionNumber := 0 , iRepetitionPeriod := 0, Comment := 'Pitch Max motor torque exceeded', Param1 := (Set:=320, SetMin:=0, SetMax:=350,Comment:='Pitch Max motor torque exceeded'), Param2 := (Set:=100, SetMin:=0, SetMax:=100,Comment:='') ),
( sName := 'a_bPitchMaxMotorCurrentExceeded', sClearName := 'Pitch Max motor current exceeded', sID := '4086', a := FALSE, b := FALSE, iGroup :=4, iSetDelay :=1, iResetDelay := 1, eResetMode := MANU, eBrakeProgram := B20, eAlarmProgram := 0, Enable := TRUE, iRepetitionNumber := 0 , iRepetitionPeriod := 0, Comment := 'Pitch Max motor current exceeded', Param1 := (Set:=70, SetMin:=28, SetMax:=80,Comment:='Pitch Max motor current exceeded'), Param2 := (Set:=19, SetMin:=0, SetMax:=20,Comment:='') ),
( sName := 'a_bPitchTrackingFault', sClearName := 'Pitch tracking fault', sID := '4087', a := FALSE, b := FALSE, iGroup :=4, iSetDelay :=10, iResetDelay := 10, eResetMode := MANU, eBrakeProgram := B20, eAlarmProgram := EMAIL, Enable := TRUE, iRepetitionNumber := 0 , iRepetitionPeriod := 10, Comment := 'Pitch tracking fault', Param1 := (Set:=2.5, SetMin:=1, SetMax:=5,Comment:=''), Param2 := (Set:=0, SetMin:=0, SetMax:=0,Comment:='') ),
( sName := 'a_bPitchTrackingWarning', sClearName := 'Pitch tracking warning', sID := '4088', a := FALSE, b := FALSE, iGroup :=4, iSetDelay :=10, iResetDelay := 10, eResetMode := MANU, eBrakeProgram := B99, eAlarmProgram := EMAIL, Enable := TRUE, iRepetitionNumber := 0 , iRepetitionPeriod := 10, Comment := 'Pitch tracking warning', Param1 := (Set:=1.5, SetMin:=1, SetMax:=3,Comment:=''), Param2 := (Set:=0, SetMin:=0, SetMax:=0,Comment:='') ),
( sName := 'a_bPitchFineSoftwareLimitSwitch', sClearName := 'Pitch system detected fine limit', sID := '4089', a := FALSE, b := FALSE, iGroup :=4, iSetDelay :=1, iResetDelay := 10, eResetMode := MANU, eBrakeProgram := B4, eAlarmProgram := 0, Enable := TRUE, iRepetitionNumber := 0 , iRepetitionPeriod := 10, Comment := 'Pitch system detected fine limit', Param1 := (Set:=0, SetMin:=0, SetMax:=360,Comment:=''), Param2 := (Set:=4, SetMin:=1, SetMax:=75,Comment:='') ),
( sName := 'a_bPitchExtremeFeatherSoftwareLimitSwitch', sClearName := 'Pitch system detected fine limit', sID := '4090', a := FALSE, b := FALSE, iGroup :=4, iSetDelay :=1, iResetDelay := 10, eResetMode := MANU, eBrakeProgram := B1, eAlarmProgram := 0, Enable := TRUE, iRepetitionNumber := 0 , iRepetitionPeriod := 10, Comment := 'Pitch system detected extreme feather limit', Param1 := (Set:=90, SetMin:=88, SetMax:=90,Comment:=''), Param2 := (Set:=87, SetMin:=87, SetMax:=88,Comment:='') ),
( sName := 'a_bPitchEncoder1Fault', sClearName := 'Pitch system Blade encoder 1', sID := '4091', a := FALSE, b := FALSE, iGroup :=4, iSetDelay :=1, iResetDelay := 1, eResetMode := MANU, eBrakeProgram := B20, eAlarmProgram := 0, Enable := TRUE, iRepetitionNumber := 0 , iRepetitionPeriod := 0, Comment := 'Pitch system Blade encoder 1', Param1 := (Set:=70, SetMin:=28, SetMax:=80,Comment:='Pitch Max motor current exceeded'), Param2 := (Set:=19, SetMin:=0, SetMax:=20,Comment:='') ),
( sName := 'a_bPitchLoadedEFCTest', sClearName := 'Pitch system loaded EFC Test', sID := '4092', a := FALSE, b := FALSE, iGroup :=4, iSetDelay :=1, iResetDelay := 100, eResetMode := MANU, eBrakeProgram := B99, eAlarmProgram := 0, Enable := TRUE, iRepetitionNumber := 0 , iRepetitionPeriod := 0, Comment := 'Pitch system loaded EFC Test', Param1 := (Set:=0, SetMin:=0, SetMax:=0,Comment:=''), Param2 := (Set:=0, SetMin:=0, SetMax:=0,Comment:='') ),
( sName := 'a_bYawDummyAlarm', sClearName := 'Water level below slip ring tripped low sensor', sID := '5001', a := FALSE, b := FALSE, iGroup :=5, iSetDelay :=50, iResetDelay := 0, eResetMode := MANU, eBrakeProgram := B99, eAlarmProgram := 0, Enable := FALSE, iRepetitionNumber := 0 , iRepetitionPeriod := 0, Comment := 'Water level below slip ring tripped low sensor at bottom of trough', Param1 := (Set:=0, SetMin:=0, SetMax:=0,Comment:=''), Param2 := (Set:=0, SetMin:=0, SetMax:=0,Comment:='') ),
( sName := 'a_bLSSDummyAlarm', sClearName := '', sID := '6002', a := FALSE, b := FALSE, iGroup :=5, iSetDelay :=50, iResetDelay := 0, eResetMode := MANU, eBrakeProgram := B100, eAlarmProgram := EMAIL, Enable := FALSE, iRepetitionNumber := 0 , iRepetitionPeriod := 0, Comment := 'Ambient temperature high at front of nacelle', Param1 := (Set:=40, SetMin:=0, SetMax:=100,Comment:=''), Param2 := (Set:=0, SetMin:=0, SetMax:=0,Comment:='') ),
( sName := 'a_bGENDummyAlarm', sClearName := '', sID := '15001', a := FALSE, b := FALSE, iGroup :=5, iSetDelay :=50, iResetDelay := 0, eResetMode := MANU, eBrakeProgram := B100, eAlarmProgram := EMAIL, Enable := FALSE, iRepetitionNumber := 0 , iRepetitionPeriod := 0, Comment := 'Ambient temperature high at front of nacelle', Param1 := (Set:=40, SetMin:=0, SetMax:=100,Comment:=''), Param2 := (Set:=0, SetMin:=0, SetMax:=0,Comment:='') ),
( sName := 'a_bGearDummyAlarm', sClearName := '', sID := '8001', a := FALSE, b := FALSE, iGroup :=5, iSetDelay :=50, iResetDelay := 0, eResetMode := MANU, eBrakeProgram := B100, eAlarmProgram := EMAIL, Enable := FALSE, iRepetitionNumber := 0 , iRepetitionPeriod := 0, Comment := 'Ambient temperature high at front of nacelle', Param1 := (Set:=40, SetMin:=0, SetMax:=100,Comment:=''), Param2 := (Set:=0, SetMin:=0, SetMax:=0,Comment:='') ),
( sName := 'a_bAuxPowerBreakerError_2S1_MainSwitch', sClearName := '2S1', sID := '9001', a := FALSE, b := FALSE, iGroup :=9, iSetDelay :=0, iResetDelay := 0, eResetMode := MANU, eBrakeProgram := B99, eAlarmProgram := 0, Enable := TRUE, iRepetitionNumber := 0 , iRepetitionPeriod := 10, Comment := 'Main Supply Switch', Param1 := (Set:=0, SetMin:=0, SetMax:=0,Comment:=''), Param2 := (Set:=0, SetMin:=0, SetMax:=0,Comment:='') ),
( sName := 'a_bAuxPowerDCbusSupply01Fault', sClearName := 'a_bAuxPowerPriDCbusSupply01Fault', sID := '9038', a := FALSE, b := FALSE, iGroup :=9, iSetDelay :=30, iResetDelay := 0, eResetMode := MANU, eBrakeProgram := B99, eAlarmProgram := 0, Enable := TRUE, iRepetitionNumber := 0 , iRepetitionPeriod := 10, Comment := '', Param1 := (Set:=0, SetMin:=0, SetMax:=0,Comment:=''), Param2 := (Set:=0, SetMin:=0, SetMax:=0,Comment:='') ),
( sName := 'a_bAuxPowerDCbusUPS1AlarmActive', sClearName := 'a_bAuxPowerPriDCbusUPS1AlarmActive', sID := '9039', a := FALSE, b := FALSE, iGroup :=9, iSetDelay :=0, iResetDelay := 0, eResetMode := MANU, eBrakeProgram := B99, eAlarmProgram := 0, Enable := TRUE, iRepetitionNumber := 0 , iRepetitionPeriod := 10, Comment := '', Param1 := (Set:=0, SetMin:=0, SetMax:=0,Comment:=''), Param2 := (Set:=0, SetMin:=0, SetMax:=0,Comment:='') ),
( sName := 'a_bAuxPowerDCbusUPS1BatteryLow', sClearName := 'a_bAuxPowerPriDCbusUPS1BatteryLow', sID := '9040', a := FALSE, b := FALSE, iGroup :=9, iSetDelay :=30, iResetDelay := 0, eResetMode := MANU, eBrakeProgram := B99, eAlarmProgram := 0, Enable := TRUE, iRepetitionNumber := 0 , iRepetitionPeriod := 10, Comment := '', Param1 := (Set:=0, SetMin:=0, SetMax:=0,Comment:=''), Param2 := (Set:=0, SetMin:=0, SetMax:=0,Comment:='') ),
( sName := 'a_bAuxPowerDCbusUPS1BatteryLifeWarning', sClearName := 'a_bAuxPowerPriDCbusUPS1BatteryLifeWarning', sID := '9041', a := FALSE, b := FALSE, iGroup :=9, iSetDelay :=0, iResetDelay := 0, eResetMode := MANU, eBrakeProgram := B99, eAlarmProgram := 0, Enable := TRUE, iRepetitionNumber := 0 , iRepetitionPeriod := 10, Comment := '', Param1 := (Set:=0, SetMin:=0, SetMax:=0,Comment:=''), Param2 := (Set:=0, SetMin:=0, SetMax:=0,Comment:='') ),
( sName := 'a_bAuxPowerDCbusUPS1BatteryLifeLoLo', sClearName := 'a_bAuxPowerPriDCbusUPS1BatteryLifeLoLo', sID := '9042', a := FALSE, b := FALSE, iGroup :=9, iSetDelay :=0, iResetDelay := 0, eResetMode := MANU, eBrakeProgram := B99, eAlarmProgram := 0, Enable := TRUE, iRepetitionNumber := 0 , iRepetitionPeriod := 10, Comment := '', Param1 := (Set:=0, SetMin:=0, SetMax:=0,Comment:=''), Param2 := (Set:=0, SetMin:=0, SetMax:=0,Comment:='') ),
( sName := 'a_bAuxPowerDCbusUPS1BatteryCharging', sClearName := 'a_bAuxPowerPriDCbusUPS1BatteryCharging', sID := '9043', a := FALSE, b := FALSE, iGroup :=9, iSetDelay :=100, iResetDelay := 0, eResetMode := MANU, eBrakeProgram := B99, eAlarmProgram := 0, Enable := TRUE, iRepetitionNumber := 0 , iRepetitionPeriod := 10, Comment := '', Param1 := (Set:=0, SetMin:=0, SetMax:=0,Comment:=''), Param2 := (Set:=0, SetMin:=0, SetMax:=0,Comment:='') ),
( sName := 'a_bAuxPowerDCbusUPS1BatteryChargingTooLong', sClearName := 'a_bAuxPowerPriDCbusUPS1BatteryChargingTooLong', sID := '9044', a := FALSE, b := FALSE, iGroup :=9, iSetDelay :=108000, iResetDelay := 0, eResetMode := MANU, eBrakeProgram := B99, eAlarmProgram := 0, Enable := TRUE, iRepetitionNumber := 0 , iRepetitionPeriod := 10, Comment := '', Param1 := (Set:=0, SetMin:=0, SetMax:=0,Comment:=''), Param2 := (Set:=0, SetMin:=0, SetMax:=0,Comment:='') ),
( sName := 'a_bAuxPowerDCbusORing01RedunFault', sClearName := 'a_bAuxPowerPriDCbusORing01RedunFault', sID := '9045', a := FALSE, b := FALSE, iGroup :=9, iSetDelay :=0, iResetDelay := 0, eResetMode := MANU, eBrakeProgram := B99, eAlarmProgram := 0, Enable := TRUE, iRepetitionNumber := 0 , iRepetitionPeriod := 10, Comment := '', Param1 := (Set:=0, SetMin:=0, SetMax:=0,Comment:=''), Param2 := (Set:=0, SetMin:=0, SetMax:=0,Comment:='') ),
( sName := 'a_bAuxPowerDCbusORing01RedunWarning', sClearName := 'a_bAuxPowerPriDCbusORing01RedunWarning', sID := '9046', a := FALSE, b := FALSE, iGroup :=9, iSetDelay :=0, iResetDelay := 0, eResetMode := MANU, eBrakeProgram := B99, eAlarmProgram := 0, Enable := TRUE, iRepetitionNumber := 0 , iRepetitionPeriod := 10, Comment := '', Param1 := (Set:=0, SetMin:=0, SetMax:=0,Comment:=''), Param2 := (Set:=0, SetMin:=0, SetMax:=0,Comment:='') ),
( sName := 'a_bAuxPowerDCbusDCVoltageLow', sClearName := '', sID := '9074', a := FALSE, b := FALSE, iGroup :=9, iSetDelay :=0, iResetDelay := 0, eResetMode := MANU, eBrakeProgram := B99, eAlarmProgram := 0, Enable := TRUE, iRepetitionNumber := 0 , iRepetitionPeriod := 10, Comment := '24VDC Bus Low Voltage Detected', Param1 := (Set:=23, SetMin:=22, SetMax:=30,Comment:='DC Bus Voltage Low'), Param2 := (Set:=0, SetMin:=0, SetMax:=0,Comment:='') ),
( sName := 'a_bStatusBackupChargerAxis1CriticalError', sClearName := 'a_bStatusBackupChargerAxis1CriticalError', sID := '9074', a := FALSE, b := FALSE, iGroup :=9, iSetDelay :=0, iResetDelay := 0, eResetMode := MANU, eBrakeProgram := B1, eAlarmProgram := 0, Enable := TRUE, iRepetitionNumber := 0 , iRepetitionPeriod := 10, Comment := 'a_bStatusBackupChargerAxis1CriticalError', Param1 := (Set:=0, SetMin:=0, SetMax:=0,Comment:=''), Param2 := (Set:=0, SetMin:=0, SetMax:=0,Comment:='') ),
( sName := 'a_bGridLossDetected', sClearName := '', sID := '10001', a := FALSE, b := FALSE, iGroup :=10, iSetDelay :=0, iResetDelay := 0, eResetMode := MANU, eBrakeProgram := B17, eAlarmProgram := 0, Enable := TRUE, iRepetitionNumber := 0 , iRepetitionPeriod := 10, Comment := 'Grid loss detected by converter', Param1 := (Set:=0, SetMin:=0, SetMax:=0,Comment:=''), Param2 := (Set:=0, SetMin:=0, SetMax:=0,Comment:='') ),
( sName := 'a_bLowVoltageRideThrough', sClearName := '', sID := '10002', a := FALSE, b := FALSE, iGroup :=10, iSetDelay :=0, iResetDelay := 0, eResetMode := MANU, eBrakeProgram := B99, eAlarmProgram := 0, Enable := TRUE, iRepetitionNumber := 0 , iRepetitionPeriod := 10, Comment := 'LVRT detected by converter', Param1 := (Set:=0, SetMin:=0, SetMax:=0,Comment:=''), Param2 := (Set:=0, SetMin:=0, SetMax:=0,Comment:='') ),
( sName := 'a_bScadaEnableAutoStartRequested', sClearName := '', sID := '11001', a := FALSE, b := FALSE, iGroup :=11, iSetDelay :=0, iResetDelay := 0, eResetMode := MANU, eBrakeProgram := B99, eAlarmProgram := 0, Enable := TRUE, iRepetitionNumber := 0 , iRepetitionPeriod := 0, Comment := 'SCADA enable autostart requested', Param1 := (Set:=0, SetMin:=0, SetMax:=0,Comment:=''), Param2 := (Set:=0, SetMin:=0, SetMax:=0,Comment:='') ),
( sName := 'a_bScadaDisableAutoStartRequested', sClearName := '', sID := '11002', a := FALSE, b := FALSE, iGroup :=11, iSetDelay :=0, iResetDelay := 0, eResetMode := MANU, eBrakeProgram := B99, eAlarmProgram := 0, Enable := TRUE, iRepetitionNumber := 0 , iRepetitionPeriod := 0, Comment := 'SCADA disable autostart requested', Param1 := (Set:=0, SetMin:=0, SetMax:=0,Comment:=''), Param2 := (Set:=0, SetMin:=0, SetMax:=0,Comment:='') ),
( sName := 'a_bScadaNormalStopRequested', sClearName := '', sID := '11003', a := FALSE, b := FALSE, iGroup :=11, iSetDelay :=0, iResetDelay := 0, eResetMode := MANU, eBrakeProgram := B99, eAlarmProgram := 0, Enable := TRUE, iRepetitionNumber := 0 , iRepetitionPeriod := 0, Comment := 'SCADA normal stop requested', Param1 := (Set:=0, SetMin:=0, SetMax:=0,Comment:=''), Param2 := (Set:=0, SetMin:=0, SetMax:=0,Comment:='') ),
( sName := 'a_bScadaAlarmResetRequested', sClearName := '', sID := '11004', a := FALSE, b := FALSE, iGroup :=11, iSetDelay :=0, iResetDelay := 0, eResetMode := MANU, eBrakeProgram := B99, eAlarmProgram := 0, Enable := TRUE, iRepetitionNumber := 0 , iRepetitionPeriod := 0, Comment := 'SCADA alarm reset requested', Param1 := (Set:=0, SetMin:=0, SetMax:=0,Comment:=''), Param2 := (Set:=0, SetMin:=0, SetMax:=0,Comment:='') ),
( sName := 'a_bScadaSafetyResetRequested', sClearName := '', sID := '11005', a := FALSE, b := FALSE, iGroup :=11, iSetDelay :=0, iResetDelay := 0, eResetMode := MANU, eBrakeProgram := B99, eAlarmProgram := 0, Enable := TRUE, iRepetitionNumber := 0 , iRepetitionPeriod := 0, Comment := 'SCADA safety reset requested', Param1 := (Set:=0, SetMin:=0, SetMax:=0,Comment:=''), Param2 := (Set:=0, SetMin:=0, SetMax:=0,Comment:='') ),
( sName := 'a_bScadaOpModeChangeRequested', sClearName := '', sID := '11006', a := FALSE, b := FALSE, iGroup :=11, iSetDelay :=0, iResetDelay := 0, eResetMode := MANU, eBrakeProgram := B99, eAlarmProgram := 0, Enable := TRUE, iRepetitionNumber := 0 , iRepetitionPeriod := 0, Comment := 'SCADA op mode change requested', Param1 := (Set:=0, SetMin:=0, SetMax:=0,Comment:=''), Param2 := (Set:=0, SetMin:=0, SetMax:=0,Comment:='') ),
( sName := 'a_bScadaServiceIdleStRequest', sClearName := '', sID := '11007', a := FALSE, b := FALSE, iGroup :=11, iSetDelay :=0, iResetDelay := 0, eResetMode := MANU, eBrakeProgram := B99, eAlarmProgram := 0, Enable := TRUE, iRepetitionNumber := 0 , iRepetitionPeriod := 0, Comment := 'SCADA service idle ST request', Param1 := (Set:=0, SetMin:=0, SetMax:=0,Comment:=''), Param2 := (Set:=0, SetMin:=0, SetMax:=0,Comment:='') ),
( sName := 'a_bScadaServiceStopStRequest', sClearName := '', sID := '11008', a := FALSE, b := FALSE, iGroup :=11, iSetDelay :=0, iResetDelay := 0, eResetMode := MANU, eBrakeProgram := B99, eAlarmProgram := 0, Enable := TRUE, iRepetitionNumber := 0 , iRepetitionPeriod := 0, Comment := 'SCADA service stop ST request', Param1 := (Set:=0, SetMin:=0, SetMax:=0,Comment:=''), Param2 := (Set:=0, SetMin:=0, SetMax:=0,Comment:='') ),
( sName := 'a_bScadaEnableSafetyNACPRequested', sClearName := '', sID := '11009', a := FALSE, b := FALSE, iGroup :=11, iSetDelay :=0, iResetDelay := 0, eResetMode := MANU, eBrakeProgram := B99, eAlarmProgram := 0, Enable := TRUE, iRepetitionNumber := 0 , iRepetitionPeriod := 0, Comment := 'SCADA enable safety NACP requested', Param1 := (Set:=0, SetMin:=0, SetMax:=0,Comment:=''), Param2 := (Set:=0, SetMin:=0, SetMax:=0,Comment:='') ),
( sName := 'a_bScadaDisableSafetyNACPRequested', sClearName := '', sID := '11010', a := FALSE, b := FALSE, iGroup :=11, iSetDelay :=0, iResetDelay := 0, eResetMode := MANU, eBrakeProgram := B99, eAlarmProgram := 0, Enable := TRUE, iRepetitionNumber := 0 , iRepetitionPeriod := 0, Comment := 'SCADA disable safety NACP requested', Param1 := (Set:=0, SetMin:=0, SetMax:=0,Comment:=''), Param2 := (Set:=0, SetMin:=0, SetMax:=0,Comment:='') ),
( sName := 'a_bScadaEnableSafetyNACSRequested', sClearName := '', sID := '11011', a := FALSE, b := FALSE, iGroup :=11, iSetDelay :=0, iResetDelay := 0, eResetMode := MANU, eBrakeProgram := B99, eAlarmProgram := 0, Enable := TRUE, iRepetitionNumber := 0 , iRepetitionPeriod := 0, Comment := 'SCADA enable safety NACS requested', Param1 := (Set:=0, SetMin:=0, SetMax:=0,Comment:=''), Param2 := (Set:=0, SetMin:=0, SetMax:=0,Comment:='') ),
( sName := 'a_bScadaDisableSafetyNACSRequested', sClearName := '', sID := '11012', a := FALSE, b := FALSE, iGroup :=11, iSetDelay :=0, iResetDelay := 0, eResetMode := MANU, eBrakeProgram := B99, eAlarmProgram := 0, Enable := TRUE, iRepetitionNumber := 0 , iRepetitionPeriod := 0, Comment := 'SCADA disable safety NACS requested', Param1 := (Set:=0, SetMin:=0, SetMax:=0,Comment:=''), Param2 := (Set:=0, SetMin:=0, SetMax:=0,Comment:='') ),
( sName := 'a_bScadaLossOfCommsToTTGC', sClearName := '', sID := '11013', a := FALSE, b := FALSE, iGroup :=11, iSetDelay :=0, iResetDelay := 0, eResetMode := MANU, eBrakeProgram := B99, eAlarmProgram := 0, Enable := TRUE, iRepetitionNumber := 0 , iRepetitionPeriod := 0, Comment := 'SCADA loss of comms to TTGC', Param1 := (Set:=0, SetMin:=0, SetMax:=0,Comment:=''), Param2 := (Set:=0, SetMin:=0, SetMax:=0,Comment:='') )];
iMaxAlarms: INT := 222;
arrAlarmStatus: ARRAY [1..222] OF BOOL;
arrAlarmGroup: ARRAY [1..222] OF INT;
END_VAR
*)


